LIN {X 0,Y 354.9,Z 351.278,A -85,B 0,C 180,E1 -13564.173,E2 -13564.173} C_VEL
LIN {X 0,Y 354.84,Z 351.284,A -85,B 0,C 180,E1 -13567.894,E2 -13567.894} C_VEL
LIN {X 0,Y 354.924,Z 351.273,A -85,B 0,C 180,E1 -13571.891,E2 -13571.891} C_VEL
LIN {X 0,Y 354.943,Z 351.273,A -85,B 0,C 180,E1 -13575.981,E2 -13575.981} C_VEL
LIN {X 0,Y 354.979,Z 351.267,A -85,B 0,C 180,E1 -13579.736,E2 -13579.736} C_VEL
LIN {X 0,Y 355.125,Z 351.247,A -85,B 0,C 180,E1 -13583.181,E2 -13583.181} C_VEL
LIN {X 0,Y 355.247,Z 351.234,A -85,B 0,C 180,E1 -13587.732,E2 -13587.732} C_VEL
LIN {X 0,Y 355.397,Z 351.218,A -85,B 0,C 180,E1 -13590,E2 -13590} C_VEL
LIN {X 0,Y 355.247,Z 351.234,A -85,B 0,C 180,E1 -13592.268,E2 -13592.268} C_VEL
LIN {X 0,Y 355.125,Z 351.247,A -85,B 0,C 180,E1 -13596.82,E2 -13596.82} C_VEL
LIN {X 0,Y 354.979,Z 351.267,A -85,B 0,C 180,E1 -13600.264,E2 -13600.264} C_VEL
LIN {X 0,Y 354.943,Z 351.272,A -85,B 0,C 180,E1 -13604.019,E2 -13604.019} C_VEL
LIN {X 0,Y 354.924,Z 351.274,A -85,B 0,C 180,E1 -13608.109,E2 -13608.109} C_VEL
LIN {X 0,Y 354.837,Z 351.284,A -85,B 0,C 180,E1 -13612.106,E2 -13612.106} C_VEL
LIN {X 0,Y 354.9,Z 351.278,A -85,B 0,C 180,E1 -13615.828,E2 -13615.828} C_VEL
LIN {X 0,Y 354.819,Z 351.289,A -85,B 0,C 180,E1 -13619.682,E2 -13619.682} C_VEL
LIN {X 0,Y 354.807,Z 351.289,A -85,B 0,C 180,E1 -13623.702,E2 -13623.702} C_VEL
LIN {X 0,Y 354.799,Z 351.287,A -85,B 0,C 180,E1 -13626.46,E2 -13626.46} C_VEL
LIN {X 0,Y 354.825,Z 351.288,A -85,B 0,C 180,E1 -13629.424,E2 -13629.424} C_VEL
LIN {X 0,Y 354.837,Z 351.285,A -85,B 0,C 180,E1 -13632.876,E2 -13632.876} C_VEL
LIN {X 0,Y 354.785,Z 351.289,A -85,B 0,C 180,E1 -13636.107,E2 -13636.107} C_VEL
LIN {X 0,Y 354.79,Z 351.293,A -85,B 0,C 180,E1 -13639.18,E2 -13639.18} C_VEL
LIN {X 0,Y 354.8,Z 351.285,A -85,B 0,C 180,E1 -13641.986,E2 -13641.986} C_VEL
LIN {X 0,Y 354.179,Z 351.369,A -85,B 0,C 180,E1 -13642.933,E2 -13642.933} C_VEL
LIN {X 0,Y 351.343,Z 351.731,A -85,B 0,C 180,E1 -13644.472,E2 -13644.472} C_VEL
LIN {X 0,Y 348.898,Z 352.035,A -85,B 0,C 180,E1 -13645.718,E2 -13645.718} C_VEL
LIN {X 0,Y 347.828,Z 352.162,A -85,B 0,C 180,E1 -13646.683,E2 -13646.683} C_VEL
LIN {X 0,Y 347.732,Z 352.171,A -85,B 0,C 180,E1 -13647.01,E2 -13647.01} C_VEL
LIN {X 0,Y 347.808,Z 352.163,A -85,B 0,C 180,E1 -13650.991,E2 -13650.991} C_VEL
LIN {X 0,Y 347.835,Z 352.155,A -85,B 0,C 180,E1 -13653.608,E2 -13653.608} C_VEL
LIN {X 0,Y 347.792,Z 352.16,A -85,B 0,C 180,E1 -13656.162,E2 -13656.162} C_VEL
LIN {X 0,Y 347.816,Z 352.156,A -85,B 0,C 180,E1 -13659.91,E2 -13659.91} C_VEL
LIN {X 0,Y 347.87,Z 352.152,A -85,B 0,C 180,E1 -13662.36,E2 -13662.36} C_VEL
LIN {X 0,Y 347.901,Z 352.147,A -85,B 0,C 180,E1 -13665.971,E2 -13665.971} C_VEL
LIN {X 0,Y 347.933,Z 352.143,A -85,B 0,C 180,E1 -13669.526,E2 -13669.526} C_VEL
LIN {X 0,Y 348.079,Z 352.125,A -85,B 0,C 180,E1 -13671.875,E2 -13671.875} C_VEL
LIN {X 0,Y 348.072,Z 352.127,A -85,B 0,C 180,E1 -13674.206,E2 -13674.206} C_VEL
LIN {X 0,Y 348.21,Z 352.107,A -85,B 0,C 180,E1 -13677.687,E2 -13677.687} C_VEL
LIN {X 0,Y 348.35,Z 352.092,A -85,B 0,C 180,E1 -13680,E2 -13680} C_VEL
LIN {X 0,Y 348.213,Z 352.112,A -85,B 0,C 180,E1 -13682.314,E2 -13682.314} C_VEL
LIN {X 0,Y 348.082,Z 352.125,A -85,B 0,C 180,E1 -13686.958,E2 -13686.958} C_VEL
LIN {X 0,Y 347.932,Z 352.147,A -85,B 0,C 180,E1 -13690.474,E2 -13690.474} C_VEL
LIN {X 0,Y 347.903,Z 352.15,A -85,B 0,C 180,E1 -13694.15,E2 -13694.15} C_VEL
LIN {X 0,Y 347.896,Z 352.151,A -85,B 0,C 180,E1 -13698.291,E2 -13698.291} C_VEL
LIN {X 0,Y 347.793,Z 352.161,A -85,B 0,C 180,E1 -13701.635,E2 -13701.635} C_VEL
LIN {X 0,Y 347.817,Z 352.157,A -85,B 0,C 180,E1 -13705.108,E2 -13705.108} C_VEL
LIN {X 0,Y 347.815,Z 352.16,A -85,B 0,C 180,E1 -13707.694,E2 -13707.694} C_VEL
LIN {X 0,Y 347.768,Z 352.165,A -85,B 0,C 180,E1 -13710.346,E2 -13710.346} C_VEL
LIN {X 0,Y 347.748,Z 352.166,A -85,B 0,C 180,E1 -13714.464,E2 -13714.464} C_VEL
LIN {X 0,Y 347.778,Z 352.166,A -85,B 0,C 180,E1 -13717.989,E2 -13717.989} C_VEL
LIN {X 0,Y 347.754,Z 352.169,A -85,B 0,C 180,E1 -13721.83,E2 -13721.83} C_VEL
LIN {X 0,Y 347.796,Z 352.242,A -85,B 0,C 180,E1 -13724.098,E2 -13724.098} C_VEL
LIN {X 0,Y 349.366,Z 360.314,A -85,B 0,C 180,E1 -13727.345,E2 -13727.345} C_VEL
LIN {X 0,Y 351.389,Z 370.514,A -85,B 0,C 180,E1 -13731.263,E2 -13731.263} C_VEL
LIN {X 0,Y 351.886,Z 373.789,A -85,B 0,C 180,E1 -13732.472,E2 -13732.472} C_VEL
LIN {X 0,Y 350.707,Z 383.556,A -85,B 0,C 180,E1 -13735.867,E2 -13735.867} C_VEL
LIN {X 0,Y 349.465,Z 395.227,A -85,B 0,C 180,E1 -13739.856,E2 -13739.856} C_VEL
LIN {X 0,Y 348.417,Z 406.538,A -85,B 0,C 180,E1 -13743.655,E2 -13743.655} C_VEL
LIN {X 0,Y 347.759,Z 415.945,A -85,B 0,C 180,E1 -13746.791,E2 -13746.791} C_VEL
LIN {X 0,Y 347.166,Z 427.344,A -85,B 0,C 180,E1 -13750.563,E2 -13750.563} C_VEL
LIN {X 0,Y 348.118,Z 441.877,A -85,B 0,C 180,E1 -13751.226,E2 -13751.226} C_VEL
LIN {X 0,Y 349.033,Z 455.463,A -85,B 0,C 180,E1 -13752.084,E2 -13752.084} C_VEL
LIN {X 0,Y 349.717,Z 469.057,A -85,B 0,C 180,E1 -13753.209,E2 -13753.209} C_VEL
LIN {X 0,Y 349.808,Z 475.163,A -85,B 0,C 180,E1 -13753.813,E2 -13753.813} C_VEL
LIN {X 0,Y 348.741,Z 487.264,A -85,B 0,C 180,E1 -13755.234,E2 -13755.234} C_VEL
LIN {X 0,Y 348.022,Z 496.484,A -85,B 0,C 180,E1 -13756.571,E2 -13756.571} C_VEL
LIN {X 0,Y 347.479,Z 504.803,A -85,B 0,C 180,E1 -13758.035,E2 -13758.035} C_VEL
LIN {X 0,Y 347.098,Z 512.961,A -85,B 0,C 180,E1 -13759.795,E2 -13759.795} C_VEL
LIN {X 0,Y 347.02,Z 518.533,A -85,B 0,C 180,E1 -13761.263,E2 -13761.263} C_VEL
LIN {X 0,Y 347.078,Z 523.927,A -85,B 0,C 180,E1 -13763.022,E2 -13763.022} C_VEL
LIN {X 0,Y 347.314,Z 528.073,A -85,B 0,C 180,E1 -13764.775,E2 -13764.775} C_VEL
LIN {X 0,Y 347.398,Z 531.023,A -85,B 0,C 180,E1 -13766.52,E2 -13766.52} C_VEL
LIN {X 0,Y 347.478,Z 532.411,A -85,B 0,C 180,E1 -13767.682,E2 -13767.682} C_VEL
LIN {X 0,Y 347.68,Z 533.326,A -85,B 0,C 180,E1 -13768.842,E2 -13768.842} C_VEL
LIN {X 0,Y 347.825,Z 533.775,A -85,B 0,C 180,E1 -13770,E2 -13770} C_VEL
LIN {X 0,Y 347.632,Z 533.739,A -85,B 0,C 180,E1 -13771.158,E2 -13771.158} C_VEL
LIN {X 0,Y 347.338,Z 533.253,A -85,B 0,C 180,E1 -13772.319,E2 -13772.319} C_VEL
LIN {X 0,Y 347.249,Z 532.323,A -85,B 0,C 180,E1 -13773.481,E2 -13773.481} C_VEL
LIN {X 0,Y 347.148,Z 530.952,A -85,B 0,C 180,E1 -13774.645,E2 -13774.645} C_VEL
LIN {X 0,Y 346.816,Z 527.255,A -85,B 0,C 180,E1 -13776.803,E2 -13776.803} C_VEL
LIN {X 0,Y 346.748,Z 522.608,A -85,B 0,C 180,E1 -13778.744,E2 -13778.744} C_VEL
LIN {X 0,Y 346.991,Z 516.19,A -85,B 0,C 180,E1 -13780.798,E2 -13780.798} C_VEL
LIN {X 0,Y 347.662,Z 508.139,A -85,B 0,C 180,E1 -13782.848,E2 -13782.848} C_VEL
LIN {X 0,Y 348.606,Z 499.648,A -85,B 0,C 180,E1 -13784.602,E2 -13784.602} C_VEL
LIN {X 0,Y 350.109,Z 489.465,A -85,B 0,C 180,E1 -13786.322,E2 -13786.322} C_VEL
LIN {X 0,Y 351.852,Z 478.234,A -85,B 0,C 180,E1 -13787.885,E2 -13787.885} C_VEL
LIN {X 0,Y 352.667,Z 465.91,A -85,B 0,C 180,E1 -13789.348,E2 -13789.348} C_VEL
LIN {X 0,Y 353.333,Z 454.376,A -85,B 0,C 180,E1 -13790.502,E2 -13790.502} C_VEL
LIN {X 0,Y 352.981,Z 441.435,A -85,B 0,C 180,E1 -13791.675,E2 -13791.675} C_VEL
LIN {X 0,Y 351.394,Z 428.535,A -85,B 0,C 180,E1 -13792.778,E2 -13792.778} C_VEL
LIN {X 0,Y 348.621,Z 415.219,A -85,B 0,C 180,E1 -13793.896,E2 -13793.896} C_VEL
LIN {X 0,Y 347.813,Z 411.035,A -85,B 0,C 180,E1 -13794.239,E2 -13794.239} C_VEL
LIN {X 0,Y 348.505,Z 400.916,A -85,B 0,C 180,E1 -13797.634,E2 -13797.634} C_VEL
LIN {X 0,Y 349.397,Z 391.787,A -85,B 0,C 180,E1 -13800.859,E2 -13800.859} C_VEL
LIN {X 0,Y 350.778,Z 381.485,A -85,B 0,C 180,E1 -13804.769,E2 -13804.769} C_VEL
LIN {X 0,Y 352.109,Z 374.816,A -85,B 0,C 180,E1 -13807.503,E2 -13807.503} C_VEL
LIN {X 0,Y 351.539,Z 370.215,A -85,B 0,C 180,E1 -13809.773,E2 -13809.773} C_VEL
LIN {X 0,Y 350.498,Z 364.605,A -85,B 0,C 180,E1 -13812.981,E2 -13812.981} C_VEL
LIN {X 0,Y 349.381,Z 359.714,A -85,B 0,C 180,E1 -13816.399,E2 -13816.399} C_VEL
LIN {X 0,Y 348.924,Z 357.382,A -85,B 0,C 180,E1 -13818.342,E2 -13818.342} C_VEL
LIN {X 0,Y 348.163,Z 353.938,A -85,B 0,C 180,E1 -13821.93,E2 -13821.93} C_VEL
LIN {X 0,Y 347.798,Z 352.163,A -85,B 0,C 180,E1 -13824.482,E2 -13824.482} C_VEL
LIN {X 0,Y 347.748,Z 352.166,A -85,B 0,C 180,E1 -13828.3,E2 -13828.3} C_VEL
LIN {X 0,Y 347.808,Z 352.161,A -85,B 0,C 180,E1 -13830.99,E2 -13830.99} C_VEL
LIN {X 0,Y 347.835,Z 352.156,A -85,B 0,C 180,E1 -13833.608,E2 -13833.608} C_VEL
LIN {X 0,Y 347.843,Z 352.27,A -85,B 0,C 180,E1 -13835.277,E2 -13835.277} C_VEL
LIN {X 0,Y 348.889,Z 355.097,A -85,B 0,C 180,E1 -13835.649,E2 -13835.649} C_VEL
LIN {X 0,Y 349.761,Z 356.218,A -85,B 0,C 180,E1 -13835.875,E2 -13835.875} C_VEL
LIN {X 0,Y 355.432,Z 368.089,A -85,B 0,C 180,E1 -13837.74,E2 -13837.74} C_VEL
LIN {X 0,Y 358.834,Z 377.479,A -85,B 0,C 180,E1 -13839.196,E2 -13839.196} C_VEL
LIN {X 0,Y 359.888,Z 381.885,A -85,B 0,C 180,E1 -13839.87,E2 -13839.87} C_VEL
LIN {X 0,Y 358.454,Z 392.191,A -85,B 0,C 180,E1 -13841.125,E2 -13841.125} C_VEL
LIN {X 0,Y 356.868,Z 401.532,A -85,B 0,C 180,E1 -13842.523,E2 -13842.523} C_VEL
LIN {X 0,Y 355.192,Z 410.63,A -85,B 0,C 180,E1 -13844.213,E2 -13844.213} C_VEL
LIN {X 0,Y 353.658,Z 418.033,A -85,B 0,C 180,E1 -13845.91,E2 -13845.91} C_VEL
LIN {X 0,Y 352.237,Z 424.697,A -85,B 0,C 180,E1 -13847.871,E2 -13847.871} C_VEL
LIN {X 0,Y 351.047,Z 429.307,A -85,B 0,C 180,E1 -13849.62,E2 -13849.62} C_VEL
LIN {X 0,Y 350.364,Z 431.687,A -85,B 0,C 180,E1 -13850.765,E2 -13850.765} C_VEL
LIN {X 0,Y 349.862,Z 433.615,A -85,B 0,C 180,E1 -13851.916,E2 -13851.916} C_VEL
LIN {X 0,Y 349.316,Z 435.152,A -85,B 0,C 180,E1 -13853.066,E2 -13853.066} C_VEL
LIN {X 0,Y 348.965,Z 436.221,A -85,B 0,C 180,E1 -13854.22,E2 -13854.22} C_VEL
LIN {X 0,Y 348.368,Z 437.149,A -85,B 0,C 180,E1 -13856.53,E2 -13856.53} C_VEL
LIN {X 0,Y 348.165,Z 437.026,A -85,B 0,C 180,E1 -13857.686,E2 -13857.686} C_VEL
LIN {X 0,Y 348.011,Z 436.465,A -85,B 0,C 180,E1 -13858.843,E2 -13858.843} C_VEL
LIN {X 0,Y 347.933,Z 435.505,A -85,B 0,C 180,E1 -13860,E2 -13860} C_VEL
LIN {X 0,Y 347.774,Z 434.173,A -85,B 0,C 180,E1 -13861.158,E2 -13861.158} C_VEL
LIN {X 0,Y 347.754,Z 431.335,A -85,B 0,C 180,E1 -13862.896,E2 -13862.896} C_VEL
LIN {X 0,Y 347.898,Z 427.484,A -85,B 0,C 180,E1 -13864.635,E2 -13864.635} C_VEL
LIN {X 0,Y 348.373,Z 422.514,A -85,B 0,C 180,E1 -13866.37,E2 -13866.37} C_VEL
LIN {X 0,Y 348.729,Z 416.322,A -85,B 0,C 180,E1 -13868.11,E2 -13868.11} C_VEL
LIN {X 0,Y 349.305,Z 408.669,A -85,B 0,C 180,E1 -13869.846,E2 -13869.846} C_VEL
LIN {X 0,Y 349.935,Z 399.29,A -85,B 0,C 180,E1 -13871.586,E2 -13871.586} C_VEL
LIN {X 0,Y 350.781,Z 388.629,A -85,B 0,C 180,E1 -13873.173,E2 -13873.173} C_VEL
LIN {X 0,Y 351.477,Z 377.977,A -85,B 0,C 180,E1 -13874.474,E2 -13874.474} C_VEL
LIN {X 0,Y 351.792,Z 367.9,A -85,B 0,C 180,E1 -13875.497,E2 -13875.497} C_VEL
LIN {X 0,Y 348.726,Z 355.743,A -85,B 0,C 180,E1 -13876.614,E2 -13876.614} C_VEL
LIN {X 0,Y 347.872,Z 352.153,A -85,B 0,C 180,E1 -13876.921,E2 -13876.921} C_VEL
LIN {X 0,Y 347.814,Z 352.157,A -85,B 0,C 180,E1 -13880.09,E2 -13880.09} C_VEL
LIN {X 0,Y 347.791,Z 352.16,A -85,B 0,C 180,E1 -13883.838,E2 -13883.838} C_VEL
LIN {X 0,Y 347.854,Z 352.156,A -85,B 0,C 180,E1 -13887.255,E2 -13887.255} C_VEL
LIN {X 0,Y 347.766,Z 352.164,A -85,B 0,C 180,E1 -13890.346,E2 -13890.346} C_VEL
LIN {X 0,Y 347.746,Z 352.167,A -85,B 0,C 180,E1 -13894.464,E2 -13894.464} C_VEL
LIN {X 0,Y 347.778,Z 352.161,A -85,B 0,C 180,E1 -13897.989,E2 -13897.989} C_VEL
LIN {X 0,Y 347.768,Z 352.163,A -85,B 0,C 180,E1 -13901.828,E2 -13901.828} C_VEL
LIN {X 0,Y 347.768,Z 352.166,A -85,B 0,C 180,E1 -13905.016,E2 -13905.016} C_VEL
LIN {X 0,Y 347.752,Z 352.168,A -85,B 0,C 180,E1 -13908.397,E2 -13908.397} C_VEL
LIN {X 0,Y 347.777,Z 352.162,A -85,B 0,C 180,E1 -13912.01,E2 -13912.01} C_VEL
LIN {X 0,Y 347.745,Z 352.165,A -85,B 0,C 180,E1 -13915.536,E2 -13915.536} C_VEL
LIN {X 0,Y 347.746,Z 352.169,A -85,B 0,C 180,E1 -13918.3,E2 -13918.3} C_VEL
LIN {X 0,Y 347.779,Z 352.163,A -85,B 0,C 180,E1 -13920.988,E2 -13920.988} C_VEL
LIN {X 0,Y 347.831,Z 352.155,A -85,B 0,C 180,E1 -13923.608,E2 -13923.608} C_VEL
LIN {X 0,Y 347.79,Z 352.164,A -85,B 0,C 180,E1 -13926.162,E2 -13926.162} C_VEL
LIN {X 0,Y 347.828,Z 352.157,A -85,B 0,C 180,E1 -13929.91,E2 -13929.91} C_VEL
LIN {X 0,Y 347.868,Z 352.155,A -85,B 0,C 180,E1 -13932.359,E2 -13932.359} C_VEL
LIN {X 0,Y 347.898,Z 352.15,A -85,B 0,C 180,E1 -13935.971,E2 -13935.971} C_VEL
LIN {X 0,Y 347.929,Z 352.144,A -85,B 0,C 180,E1 -13939.526,E2 -13939.526} C_VEL
LIN {X 0,Y 348.091,Z 352.123,A -85,B 0,C 180,E1 -13943.042,E2 -13943.042} C_VEL
LIN {X 0,Y 348.209,Z 352.11,A -85,B 0,C 180,E1 -13947.687,E2 -13947.687} C_VEL
LIN {X 0,Y 348.346,Z 352.096,A -85,B 0,C 180,E1 -13950,E2 -13950} C_VEL
LIN {X 0,Y 348.21,Z 352.11,A -85,B 0,C 180,E1 -13952.314,E2 -13952.314} C_VEL
LIN {X 0,Y 348.091,Z 352.123,A -85,B 0,C 180,E1 -13956.958,E2 -13956.958} C_VEL
LIN {X 0,Y 347.93,Z 352.144,A -85,B 0,C 180,E1 -13960.475,E2 -13960.475} C_VEL
LIN {X 0,Y 347.899,Z 352.149,A -85,B 0,C 180,E1 -13964.15,E2 -13964.15} C_VEL
LIN {X 0,Y 347.892,Z 352.148,A -85,B 0,C 180,E1 -13968.291,E2 -13968.291} C_VEL
LIN {X 0,Y 347.791,Z 352.165,A -85,B 0,C 180,E1 -13971.636,E2 -13971.636} C_VEL
LIN {X 0,Y 347.813,Z 352.159,A -85,B 0,C 180,E1 -13975.109,E2 -13975.109} C_VEL
LIN {X 0,Y 347.809,Z 352.162,A -85,B 0,C 180,E1 -13977.694,E2 -13977.694} C_VEL
LIN {X 0,Y 347.75,Z 352.165,A -85,B 0,C 180,E1 -13980.348,E2 -13980.348} C_VEL
LIN {X 0,Y 347.749,Z 352.166,A -85,B 0,C 180,E1 -13984.044,E2 -13984.044} C_VEL
LIN {X 0,Y 347.763,Z 352.169,A -85,B 0,C 180,E1 -13987.321,E2 -13987.321} C_VEL
LIN {X 0,Y 347.795,Z 352.16,A -85,B 0,C 180,E1 -13990.289,E2 -13990.289} C_VEL
LIN {X 0,Y 347.788,Z 352.165,A -85,B 0,C 180,E1 -13993.399,E2 -13993.399} C_VEL
LIN {X 0,Y 347.731,Z 352.169,A -85,B 0,C 180,E1 -13996.686,E2 -13996.686} C_VEL
LIN {X 0,Y 347.749,Z 352.165,A -85,B 0,C 180,E1 -14000.173,E2 -14000.173} C_VEL
LIN {X 0,Y 347.764,Z 352.165,A -85,B 0,C 180,E1 -14002.68,E2 -14002.68} C_VEL
LIN {X 0,Y 347.751,Z 352.165,A -85,B 0,C 180,E1 -14005.957,E2 -14005.957} C_VEL
LIN {X 0,Y 347.732,Z 352.171,A -85,B 0,C 180,E1 -14007.01,E2 -14007.01} C_VEL
LIN {X 0,Y 347.039,Z 352.254,A -85,B 0,C 180,E1 -14007.978,E2 -14007.978} C_VEL
LIN {X 0,Y 344.186,Z 352.61,A -85,B 0,C 180,E1 -14009.553,E2 -14009.553} C_VEL
LIN {X 0,Y 341.809,Z 352.91,A -85,B 0,C 180,E1 -14010.828,E2 -14010.828} C_VEL
LIN {X 0,Y 340.822,Z 353.028,A -85,B 0,C 180,E1 -14011.815,E2 -14011.815} C_VEL
LIN {X 0,Y 340.758,Z 353.036,A -85,B 0,C 180,E1 -14012.148,E2 -14012.148} C_VEL
LIN {X 0,Y 340.759,Z 353.036,A -85,B 0,C 180,E1 -14015.639,E2 -14015.639} C_VEL
LIN {X 0,Y 340.756,Z 353.037,A -85,B 0,C 180,E1 -14019.475,E2 -14019.475} C_VEL
LIN {X 0,Y 340.861,Z 353.023,A -85,B 0,C 180,E1 -14021.985,E2 -14021.985} C_VEL
LIN {X 0,Y 340.873,Z 353.022,A -85,B 0,C 180,E1 -14025.705,E2 -14025.705} C_VEL
LIN {X 0,Y 340.876,Z 353.022,A -85,B 0,C 180,E1 -14029.307,E2 -14029.307} C_VEL
LIN {X 0,Y 341.081,Z 352.999,A -85,B 0,C 180,E1 -14032.899,E2 -14032.899} C_VEL
LIN {X 0,Y 341.172,Z 352.984,A -85,B 0,C 180,E1 -14037.639,E2 -14037.639} C_VEL
LIN {X 0,Y 341.3,Z 352.97,A -85,B 0,C 180,E1 -14040,E2 -14040} C_VEL
LIN {X 0,Y 341.175,Z 352.989,A -85,B 0,C 180,E1 -14042.361,E2 -14042.361} C_VEL
LIN {X 0,Y 341.05,Z 353,A -85,B 0,C 180,E1 -14047.103,E2 -14047.103} C_VEL
LIN {X 0,Y 340.875,Z 353.024,A -85,B 0,C 180,E1 -14050.694,E2 -14050.694} C_VEL
LIN {X 0,Y 340.867,Z 353.027,A -85,B 0,C 180,E1 -14054.325,E2 -14054.325} C_VEL
LIN {X 0,Y 340.842,Z 353.029,A -85,B 0,C 180,E1 -14058.467,E2 -14058.467} C_VEL
LIN {X 0,Y 340.758,Z 353.039,A -85,B 0,C 180,E1 -14061.857,E2 -14061.857} C_VEL
LIN {X 0,Y 340.777,Z 353.036,A -85,B 0,C 180,E1 -14065.664,E2 -14065.664} C_VEL
LIN {X 0,Y 340.745,Z 353.041,A -85,B 0,C 180,E1 -14068.32,E2 -14068.32} C_VEL
LIN {X 0,Y 340.708,Z 353.042,A -85,B 0,C 180,E1 -14071.044,E2 -14071.044} C_VEL
LIN {X 0,Y 340.722,Z 353.041,A -85,B 0,C 180,E1 -14075.279,E2 -14075.279} C_VEL
LIN {X 0,Y 340.714,Z 353.043,A -85,B 0,C 180,E1 -14078.386,E2 -14078.386} C_VEL
LIN {X 0,Y 340.705,Z 353.047,A -85,B 0,C 180,E1 -14082.046,E2 -14082.046} C_VEL
LIN {X 0,Y 340.741,Z 353.14,A -85,B 0,C 180,E1 -14083.835,E2 -14083.835} C_VEL
LIN {X 0,Y 342.524,Z 362.377,A -85,B 0,C 180,E1 -14087.618,E2 -14087.618} C_VEL
LIN {X 0,Y 344.203,Z 370.698,A -85,B 0,C 180,E1 -14090.886,E2 -14090.886} C_VEL
LIN {X 0,Y 344.84,Z 374.465,A -85,B 0,C 180,E1 -14092.308,E2 -14092.308} C_VEL
LIN {X 0,Y 343.679,Z 384.226,A -85,B 0,C 180,E1 -14095.781,E2 -14095.781} C_VEL
LIN {X 0,Y 342.485,Z 394.939,A -85,B 0,C 180,E1 -14099.527,E2 -14099.527} C_VEL
LIN {X 0,Y 341.497,Z 405.244,A -85,B 0,C 180,E1 -14103.079,E2 -14103.079} C_VEL
LIN {X 0,Y 340.635,Z 416.46,A -85,B 0,C 180,E1 -14106.92,E2 -14106.92} C_VEL
LIN {X 0,Y 340.112,Z 426.416,A -85,B 0,C 180,E1 -14110.301,E2 -14110.301} C_VEL
LIN {X 0,Y 341.079,Z 442.102,A -85,B 0,C 180,E1 -14111.056,E2 -14111.056} C_VEL
LIN {X 0,Y 341.969,Z 455.589,A -85,B 0,C 180,E1 -14111.956,E2 -14111.956} C_VEL
LIN {X 0,Y 342.601,Z 467.846,A -85,B 0,C 180,E1 -14113.003,E2 -14113.003} C_VEL
LIN {X 0,Y 342.713,Z 475.376,A -85,B 0,C 180,E1 -14113.775,E2 -14113.775} C_VEL
LIN {X 0,Y 341.665,Z 487.006,A -85,B 0,C 180,E1 -14115.192,E2 -14115.192} C_VEL
LIN {X 0,Y 340.926,Z 496.262,A -85,B 0,C 180,E1 -14116.59,E2 -14116.59} C_VEL
LIN {X 0,Y 340.391,Z 504.438,A -85,B 0,C 180,E1 -14118.084,E2 -14118.084} C_VEL
LIN {X 0,Y 340.024,Z 512.478,A -85,B 0,C 180,E1 -14119.881,E2 -14119.881} C_VEL
LIN {X 0,Y 339.999,Z 518.948,A -85,B 0,C 180,E1 -14121.68,E2 -14121.68} C_VEL
LIN {X 0,Y 340.105,Z 524.358,A -85,B 0,C 180,E1 -14123.623,E2 -14123.623} C_VEL
LIN {X 0,Y 340.332,Z 527.843,A -85,B 0,C 180,E1 -14125.262,E2 -14125.262} C_VEL
LIN {X 0,Y 340.382,Z 529.72,A -85,B 0,C 180,E1 -14126.449,E2 -14126.449} C_VEL
LIN {X 0,Y 340.483,Z 531.149,A -85,B 0,C 180,E1 -14127.634,E2 -14127.634} C_VEL
LIN {X 0,Y 340.676,Z 532.141,A -85,B 0,C 180,E1 -14128.818,E2 -14128.818} C_VEL
LIN {X 0,Y 340.813,Z 532.631,A -85,B 0,C 180,E1 -14130,E2 -14130} C_VEL
LIN {X 0,Y 340.601,Z 532.626,A -85,B 0,C 180,E1 -14131.182,E2 -14131.182} C_VEL
LIN {X 0,Y 340.303,Z 532.179,A -85,B 0,C 180,E1 -14132.367,E2 -14132.367} C_VEL
LIN {X 0,Y 340.198,Z 531.321,A -85,B 0,C 180,E1 -14133.553,E2 -14133.553} C_VEL
LIN {X 0,Y 340.079,Z 529.987,A -85,B 0,C 180,E1 -14134.742,E2 -14134.742} C_VEL
LIN {X 0,Y 339.739,Z 526.641,A -85,B 0,C 180,E1 -14136.805,E2 -14136.805} C_VEL
LIN {X 0,Y 339.679,Z 521.815,A -85,B 0,C 180,E1 -14138.927,E2 -14138.927} C_VEL
LIN {X 0,Y 339.965,Z 515.568,A -85,B 0,C 180,E1 -14141.024,E2 -14141.024} C_VEL
LIN {X 0,Y 340.683,Z 507.658,A -85,B 0,C 180,E1 -14143.116,E2 -14143.116} C_VEL
LIN {X 0,Y 341.733,Z 499.139,A -85,B 0,C 180,E1 -14144.95,E2 -14144.95} C_VEL
LIN {X 0,Y 343.284,Z 489.47,A -85,B 0,C 180,E1 -14146.656,E2 -14146.656} C_VEL
LIN {X 0,Y 345.183,Z 477.464,A -85,B 0,C 180,E1 -14148.396,E2 -14148.396} C_VEL
LIN {X 0,Y 346.158,Z 465.409,A -85,B 0,C 180,E1 -14149.881,E2 -14149.881} C_VEL
LIN {X 0,Y 346.901,Z 453.696,A -85,B 0,C 180,E1 -14151.106,E2 -14151.106} C_VEL
LIN {X 0,Y 346.586,Z 442.117,A -85,B 0,C 180,E1 -14152.224,E2 -14152.224} C_VEL
LIN {X 0,Y 345.233,Z 429.937,A -85,B 0,C 180,E1 -14153.348,E2 -14153.348} C_VEL
LIN {X 0,Y 342.129,Z 414.017,A -85,B 0,C 180,E1 -14154.786,E2 -14154.786} C_VEL
LIN {X 0,Y 341.004,Z 409.581,A -85,B 0,C 180,E1 -14155.198,E2 -14155.198} C_VEL
LIN {X 0,Y 340.97,Z 408.959,A -85,B 0,C 180,E1 -14155.28,E2 -14155.28} C_VEL
LIN {X 0,Y 341.79,Z 398.636,A -85,B 0,C 180,E1 -14158.896,E2 -14158.896} C_VEL
LIN {X 0,Y 342.826,Z 389.705,A -85,B 0,C 180,E1 -14162.209,E2 -14162.209} C_VEL
LIN {X 0,Y 344.513,Z 379.586,A -85,B 0,C 180,E1 -14166.271,E2 -14166.271} C_VEL
LIN {X 0,Y 345.246,Z 376.385,A -85,B 0,C 180,E1 -14167.64,E2 -14167.64} C_VEL
LIN {X 0,Y 344.659,Z 371.814,A -85,B 0,C 180,E1 -14169.965,E2 -14169.965} C_VEL
LIN {X 0,Y 343.814,Z 367.247,A -85,B 0,C 180,E1 -14172.618,E2 -14172.618} C_VEL
LIN {X 0,Y 342.763,Z 362.561,A -85,B 0,C 180,E1 -14175.86,E2 -14175.86} C_VEL
LIN {X 0,Y 341.875,Z 358.319,A -85,B 0,C 180,E1 -14179.519,E2 -14179.519} C_VEL
LIN {X 0,Y 341.437,Z 356.176,A -85,B 0,C 180,E1 -14181.865,E2 -14181.865} C_VEL
LIN {X 0,Y 340.828,Z 353.656,A -85,B 0,C 180,E1 -14185.57,E2 -14185.57} C_VEL
LIN {X 0,Y 340.712,Z 353.042,A -85,B 0,C 180,E1 -14186.864,E2 -14186.864} C_VEL
LIN {X 0,Y 340.778,Z 353.033,A -85,B 0,C 180,E1 -14190.332,E2 -14190.332} C_VEL
LIN {X 0,Y 340.77,Z 353.038,A -85,B 0,C 180,E1 -14194.13,E2 -14194.13} C_VEL
LIN {X 0,Y 341.257,Z 354.834,A -85,B 0,C 180,E1 -14194.374,E2 -14194.374} C_VEL
LIN {X 0,Y 343.025,Z 357.39,A -85,B 0,C 180,E1 -14194.882,E2 -14194.882} C_VEL
LIN {X 0,Y 348.655,Z 368.859,A -85,B 0,C 180,E1 -14196.847,E2 -14196.847} C_VEL
LIN {X 0,Y 352.112,Z 377.872,A -85,B 0,C 180,E1 -14198.348,E2 -14198.348} C_VEL
LIN {X 0,Y 353.825,Z 384.581,A -85,B 0,C 180,E1 -14199.432,E2 -14199.432} C_VEL
LIN {X 0,Y 352.139,Z 394.973,A -85,B 0,C 180,E1 -14200.773,E2 -14200.773} C_VEL
LIN {X 0,Y 350.171,Z 405.658,A -85,B 0,C 180,E1 -14202.479,E2 -14202.479} C_VEL
LIN {X 0,Y 348.377,Z 414.184,A -85,B 0,C 180,E1 -14204.196,E2 -14204.196} C_VEL
LIN {X 0,Y 346.79,Z 421.072,A -85,B 0,C 180,E1 -14205.925,E2 -14205.925} C_VEL
LIN {X 0,Y 345.536,Z 426.547,A -85,B 0,C 180,E1 -14207.652,E2 -14207.652} C_VEL
LIN {X 0,Y 344.261,Z 430.973,A -85,B 0,C 180,E1 -14209.413,E2 -14209.413} C_VEL
LIN {X 0,Y 343.559,Z 433.259,A -85,B 0,C 180,E1 -14210.581,E2 -14210.581} C_VEL
LIN {X 0,Y 343.017,Z 435.102,A -85,B 0,C 180,E1 -14211.754,E2 -14211.754} C_VEL
LIN {X 0,Y 342.433,Z 436.548,A -85,B 0,C 180,E1 -14212.926,E2 -14212.926} C_VEL
LIN {X 0,Y 341.674,Z 438.125,A -85,B 0,C 180,E1 -14215.28,E2 -14215.28} C_VEL
LIN {X 0,Y 341.38,Z 438.342,A -85,B 0,C 180,E1 -14216.459,E2 -14216.459} C_VEL
LIN {X 0,Y 341.156,Z 438.132,A -85,B 0,C 180,E1 -14217.638,E2 -14217.638} C_VEL
LIN {X 0,Y 340.91,Z 436.486,A -85,B 0,C 180,E1 -14220,E2 -14220} C_VEL
LIN {X 0,Y 340.748,Z 435.083,A -85,B 0,C 180,E1 -14221.182,E2 -14221.182} C_VEL
LIN {X 0,Y 340.72,Z 432.144,A -85,B 0,C 180,E1 -14222.956,E2 -14222.956} C_VEL
LIN {X 0,Y 340.873,Z 428.189,A -85,B 0,C 180,E1 -14224.73,E2 -14224.73} C_VEL
LIN {X 0,Y 341.361,Z 423.089,A -85,B 0,C 180,E1 -14226.502,E2 -14226.502} C_VEL
LIN {X 0,Y 341.877,Z 415.678,A -85,B 0,C 180,E1 -14228.538,E2 -14228.538} C_VEL
LIN {X 0,Y 342.412,Z 407.652,A -85,B 0,C 180,E1 -14230.316,E2 -14230.316} C_VEL
LIN {X 0,Y 343.121,Z 397.528,A -85,B 0,C 180,E1 -14232.119,E2 -14232.119} C_VEL
LIN {X 0,Y 343.896,Z 387.391,A -85,B 0,C 180,E1 -14233.593,E2 -14233.593} C_VEL
LIN {X 0,Y 344.631,Z 376.16,A -85,B 0,C 180,E1 -14234.919,E2 -14234.919} C_VEL
LIN {X 0,Y 344.728,Z 368.818,A -85,B 0,C 180,E1 -14235.668,E2 -14235.668} C_VEL
LIN {X 0,Y 341.683,Z 356.599,A -85,B 0,C 180,E1 -14236.813,E2 -14236.813} C_VEL
LIN {X 0,Y 340.838,Z 353.031,A -85,B 0,C 180,E1 -14237.126,E2 -14237.126} C_VEL
LIN {X 0,Y 340.755,Z 353.037,A -85,B 0,C 180,E1 -14240.525,E2 -14240.525} C_VEL
LIN {X 0,Y 340.759,Z 353.036,A -85,B 0,C 180,E1 -14244.361,E2 -14244.361} C_VEL
LIN {X 0,Y 340.781,Z 353.035,A -85,B 0,C 180,E1 -14247.526,E2 -14247.526} C_VEL
LIN {X 0,Y 340.706,Z 353.048,A -85,B 0,C 180,E1 -14251.044,E2 -14251.044} C_VEL
LIN {X 0,Y 340.72,Z 353.043,A -85,B 0,C 180,E1 -14255.278,E2 -14255.278} C_VEL
LIN {X 0,Y 340.72,Z 353.042,A -85,B 0,C 180,E1 -14258.388,E2 -14258.388} C_VEL
LIN {X 0,Y 340.734,Z 353.039,A -85,B 0,C 180,E1 -14262.052,E2 -14262.052} C_VEL
LIN {X 0,Y 340.685,Z 353.046,A -85,B 0,C 180,E1 -14265.461,E2 -14265.461} C_VEL
LIN {X 0,Y 340.687,Z 353.05,A -85,B 0,C 180,E1 -14268.69,E2 -14268.69} C_VEL
LIN {X 0,Y 340.736,Z 353.039,A -85,B 0,C 180,E1 -14271.773,E2 -14271.773} C_VEL
LIN {X 0,Y 340.723,Z 353.04,A -85,B 0,C 180,E1 -14275.595,E2 -14275.595} C_VEL
LIN {X 0,Y 340.698,Z 353.045,A -85,B 0,C 180,E1 -14278.955,E2 -14278.955} C_VEL
LIN {X 0,Y 340.804,Z 353.031,A -85,B 0,C 180,E1 -14283.02,E2 -14283.02} C_VEL
LIN {X 0,Y 340.731,Z 353.04,A -85,B 0,C 180,E1 -14286.927,E2 -14286.927} C_VEL
LIN {X 0,Y 340.8,Z 353.032,A -85,B 0,C 180,E1 -14290.734,E2 -14290.734} C_VEL
LIN {X 0,Y 340.787,Z 353.032,A -85,B 0,C 180,E1 -14293.219,E2 -14293.219} C_VEL
LIN {X 0,Y 340.845,Z 353.026,A -85,B 0,C 180,E1 -14296.89,E2 -14296.89} C_VEL
LIN {X 0,Y 340.914,Z 353.019,A -85,B 0,C 180,E1 -14300.507,E2 -14300.507} C_VEL
LIN {X 0,Y 341.059,Z 352.999,A -85,B 0,C 180,E1 -14302.898,E2 -14302.898} C_VEL
LIN {X 0,Y 341.171,Z 352.987,A -85,B 0,C 180,E1 -14307.639,E2 -14307.639} C_VEL
LIN {X 0,Y 341.296,Z 352.974,A -85,B 0,C 180,E1 -14310,E2 -14310} C_VEL
LIN {X 0,Y 341.171,Z 352.987,A -85,B 0,C 180,E1 -14312.361,E2 -14312.361} C_VEL
LIN {X 0,Y 341.059,Z 352.999,A -85,B 0,C 180,E1 -14317.102,E2 -14317.102} C_VEL
LIN {X 0,Y 340.872,Z 353.022,A -85,B 0,C 180,E1 -14320.694,E2 -14320.694} C_VEL
LIN {X 0,Y 340.864,Z 353.024,A -85,B 0,C 180,E1 -14324.325,E2 -14324.325} C_VEL
LIN {X 0,Y 340.839,Z 353.026,A -85,B 0,C 180,E1 -14328.467,E2 -14328.467} C_VEL
LIN {X 0,Y 340.754,Z 353.04,A -85,B 0,C 180,E1 -14331.857,E2 -14331.857} C_VEL
LIN {X 0,Y 340.773,Z 353.039,A -85,B 0,C 180,E1 -14335.665,E2 -14335.665} C_VEL
LIN {X 0,Y 340.729,Z 353.04,A -85,B 0,C 180,E1 -14338.321,E2 -14338.321} C_VEL
LIN {X 0,Y 340.699,Z 353.045,A -85,B 0,C 180,E1 -14341.045,E2 -14341.045} C_VEL
LIN {X 0,Y 340.719,Z 353.045,A -85,B 0,C 180,E1 -14345.279,E2 -14345.279} C_VEL
LIN {X 0,Y 340.713,Z 353.041,A -85,B 0,C 180,E1 -14348.387,E2 -14348.387} C_VEL
LIN {X 0,Y 340.727,Z 353.045,A -85,B 0,C 180,E1 -14351.304,E2 -14351.304} C_VEL
LIN {X 0,Y 340.723,Z 353.041,A -85,B 0,C 180,E1 -14354.533,E2 -14354.533} C_VEL
LIN {X 0,Y 340.688,Z 353.046,A -85,B 0,C 180,E1 -14358.691,E2 -14358.691} C_VEL
LIN {X 0,Y 340.735,Z 353.039,A -85,B 0,C 180,E1 -14361.773,E2 -14361.773} C_VEL
LIN {X 0,Y 340.725,Z 353.041,A -85,B 0,C 180,E1 -14365.596,E2 -14365.596} C_VEL
LIN {X 0,Y 340.707,Z 353.048,A -85,B 0,C 180,E1 -14368.956,E2 -14368.956} C_VEL
LIN {X 0,Y 340.758,Z 353.036,A -85,B 0,C 180,E1 -14372.148,E2 -14372.148} C_VEL
LIN {X 0,Y 340.121,Z 353.119,A -85,B 0,C 180,E1 -14373.135,E2 -14373.135} C_VEL
LIN {X 0,Y 337.231,Z 353.479,A -85,B 0,C 180,E1 -14374.738,E2 -14374.738} C_VEL
LIN {X 0,Y 334.774,Z 353.781,A -85,B 0,C 180,E1 -14376.037,E2 -14376.037} C_VEL
LIN {X 0,Y 333.744,Z 353.914,A -85,B 0,C 180,E1 -14377.043,E2 -14377.043} C_VEL
LIN {X 0,Y 333.674,Z 353.916,A -85,B 0,C 180,E1 -14377.384,E2 -14377.384} C_VEL
LIN {X 0,Y 333.797,Z 353.903,A -85,B 0,C 180,E1 -14381.59,E2 -14381.59} C_VEL
LIN {X 0,Y 333.812,Z 353.901,A -85,B 0,C 180,E1 -14385.577,E2 -14385.577} C_VEL
LIN {X 0,Y 333.838,Z 353.9,A -85,B 0,C 180,E1 -14389.078,E2 -14389.078} C_VEL
LIN {X 0,Y 334.03,Z 353.878,A -85,B 0,C 180,E1 -14392.748,E2 -14392.748} C_VEL
LIN {X 0,Y 333.813,Z 353.902,A -85,B 0,C 180,E1 -14395.169,E2 -14395.169} C_VEL
LIN {X 0,Y 334.109,Z 353.864,A -85,B 0,C 180,E1 -14397.589,E2 -14397.589} C_VEL
LIN {X 0,Y 334.251,Z 353.848,A -85,B 0,C 180,E1 -14400,E2 -14400} C_VEL
LIN {X 0,Y 334.112,Z 353.869,A -85,B 0,C 180,E1 -14402.411,E2 -14402.411} C_VEL
LIN {X 0,Y 334.013,Z 353.879,A -85,B 0,C 180,E1 -14406.039,E2 -14406.039} C_VEL
LIN {X 0,Y 333.853,Z 353.897,A -85,B 0,C 180,E1 -14409.696,E2 -14409.696} C_VEL
LIN {X 0,Y 333.801,Z 353.902,A -85,B 0,C 180,E1 -14413.391,E2 -14413.391} C_VEL
LIN {X 0,Y 333.751,Z 353.908,A -85,B 0,C 180,E1 -14417.146,E2 -14417.146} C_VEL
LIN {X 0,Y 333.744,Z 353.911,A -85,B 0,C 180,E1 -14419.69,E2 -14419.69} C_VEL
LIN {X 0,Y 333.696,Z 353.92,A -85,B 0,C 180,E1 -14422.278,E2 -14422.278} C_VEL
LIN {X 0,Y 333.74,Z 353.914,A -85,B 0,C 180,E1 -14426.246,E2 -14426.246} C_VEL
LIN {X 0,Y 333.715,Z 353.913,A -85,B 0,C 180,E1 -14428.972,E2 -14428.972} C_VEL
LIN {X 0,Y 333.65,Z 353.922,A -85,B 0,C 180,E1 -14432.588,E2 -14432.588} C_VEL
LIN {X 0,Y 333.68,Z 353.921,A -85,B 0,C 180,E1 -14436.139,E2 -14436.139} C_VEL
LIN {X 0,Y 333.651,Z 353.922,A -85,B 0,C 180,E1 -14439.192,E2 -14439.192} C_VEL
LIN {X 0,Y 333.666,Z 353.924,A -85,B 0,C 180,E1 -14443.213,E2 -14443.213} C_VEL
LIN {X 0,Y 333.697,Z 354.141,A -85,B 0,C 180,E1 -14443.617,E2 -14443.617} C_VEL
LIN {X 0,Y 335.366,Z 362.616,A -85,B 0,C 180,E1 -14447.178,E2 -14447.178} C_VEL
LIN {X 0,Y 337.228,Z 371.946,A -85,B 0,C 180,E1 -14450.913,E2 -14450.913} C_VEL
LIN {X 0,Y 337.798,Z 375.375,A -85,B 0,C 180,E1 -14452.242,E2 -14452.242} C_VEL
LIN {X 0,Y 336.65,Z 384.836,A -85,B 0,C 180,E1 -14455.69,E2 -14455.69} C_VEL
LIN {X 0,Y 335.31,Z 396.333,A -85,B 0,C 180,E1 -14459.799,E2 -14459.799} C_VEL
LIN {X 0,Y 334.193,Z 407.642,A -85,B 0,C 180,E1 -14463.792,E2 -14463.792} C_VEL
LIN {X 0,Y 333.387,Z 418.806,A -85,B 0,C 180,E1 -14467.7,E2 -14467.7} C_VEL
LIN {X 0,Y 333.063,Z 425.596,A -85,B 0,C 180,E1 -14470.067,E2 -14470.067} C_VEL
LIN {X 0,Y 333.913,Z 440.603,A -85,B 0,C 180,E1 -14470.797,E2 -14470.797} C_VEL
LIN {X 0,Y 334.773,Z 454.323,A -85,B 0,C 180,E1 -14471.724,E2 -14471.724} C_VEL
LIN {X 0,Y 335.448,Z 466.517,A -85,B 0,C 180,E1 -14472.786,E2 -14472.786} C_VEL
LIN {X 0,Y 335.6,Z 475.492,A -85,B 0,C 180,E1 -14473.734,E2 -14473.734} C_VEL
LIN {X 0,Y 334.641,Z 485.822,A -85,B 0,C 180,E1 -14475.034,E2 -14475.034} C_VEL
LIN {X 0,Y 333.834,Z 495.949,A -85,B 0,C 180,E1 -14476.61,E2 -14476.61} C_VEL
LIN {X 0,Y 333.313,Z 503.999,A -85,B 0,C 180,E1 -14478.136,E2 -14478.136} C_VEL
LIN {X 0,Y 332.985,Z 511.931,A -85,B 0,C 180,E1 -14479.972,E2 -14479.972} C_VEL
LIN {X 0,Y 332.954,Z 517.306,A -85,B 0,C 180,E1 -14481.503,E2 -14481.503} C_VEL
LIN {X 0,Y 333.091,Z 522.957,A -85,B 0,C 180,E1 -14483.516,E2 -14483.516} C_VEL
LIN {X 0,Y 333.305,Z 526.454,A -85,B 0,C 180,E1 -14485.162,E2 -14485.162} C_VEL
LIN {X 0,Y 333.365,Z 528.399,A -85,B 0,C 180,E1 -14486.374,E2 -14486.374} C_VEL
LIN {X 0,Y 333.484,Z 529.872,A -85,B 0,C 180,E1 -14487.584,E2 -14487.584} C_VEL
LIN {X 0,Y 333.671,Z 530.91,A -85,B 0,C 180,E1 -14488.793,E2 -14488.793} C_VEL
LIN {X 0,Y 333.802,Z 531.476,A -85,B 0,C 180,E1 -14490,E2 -14490} C_VEL
LIN {X 0,Y 333.595,Z 531.512,A -85,B 0,C 180,E1 -14491.207,E2 -14491.207} C_VEL
LIN {X 0,Y 333.146,Z 530.289,A -85,B 0,C 180,E1 -14493.628,E2 -14493.628} C_VEL
LIN {X 0,Y 333.011,Z 529.03,A -85,B 0,C 180,E1 -14494.842,E2 -14494.842} C_VEL
LIN {X 0,Y 332.646,Z 525.136,A -85,B 0,C 180,E1 -14497.283,E2 -14497.283} C_VEL
LIN {X 0,Y 332.599,Z 521.045,A -85,B 0,C 180,E1 -14499.119,E2 -14499.119} C_VEL
LIN {X 0,Y 332.831,Z 515.9,A -85,B 0,C 180,E1 -14500.955,E2 -14500.955} C_VEL
LIN {X 0,Y 333.563,Z 508.452,A -85,B 0,C 180,E1 -14503.091,E2 -14503.091} C_VEL
LIN {X 0,Y 334.769,Z 499.447,A -85,B 0,C 180,E1 -14505.151,E2 -14505.151} C_VEL
LIN {X 0,Y 336.491,Z 489.525,A -85,B 0,C 180,E1 -14507.002,E2 -14507.002} C_VEL
LIN {X 0,Y 338.357,Z 478.935,A -85,B 0,C 180,E1 -14508.624,E2 -14508.624} C_VEL
LIN {X 0,Y 339.404,Z 467.565,A -85,B 0,C 180,E1 -14510.136,E2 -14510.136} C_VEL
LIN {X 0,Y 340.445,Z 455.223,A -85,B 0,C 180,E1 -14511.526,E2 -14511.526} C_VEL
LIN {X 0,Y 340.277,Z 443.048,A -85,B 0,C 180,E1 -14512.784,E2 -14512.784} C_VEL
LIN {X 0,Y 339.178,Z 431.524,A -85,B 0,C 180,E1 -14513.926,E2 -14513.926} C_VEL
LIN {X 0,Y 336.459,Z 416.697,A -85,B 0,C 180,E1 -14515.389,E2 -14515.389} C_VEL
LIN {X 0,Y 335.009,Z 411.047,A -85,B 0,C 180,E1 -14515.973,E2 -14515.973} C_VEL
LIN {X 0,Y 334.186,Z 406.936,A -85,B 0,C 180,E1 -14516.376,E2 -14516.376} C_VEL
LIN {X 0,Y 335.375,Z 394.983,A -85,B 0,C 180,E1 -14520.775,E2 -14520.775} C_VEL
LIN {X 0,Y 336.936,Z 384.471,A -85,B 0,C 180,E1 -14524.968,E2 -14524.968} C_VEL
LIN {X 0,Y 338.35,Z 377.774,A -85,B 0,C 180,E1 -14527.878,E2 -14527.878} C_VEL
LIN {X 0,Y 337.772,Z 373.412,A -85,B 0,C 180,E1 -14530.167,E2 -14530.167} C_VEL
LIN {X 0,Y 336.728,Z 367.907,A -85,B 0,C 180,E1 -14533.532,E2 -14533.532} C_VEL
LIN {X 0,Y 335.658,Z 363.135,A -85,B 0,C 180,E1 -14537.125,E2 -14537.125} C_VEL
LIN {X 0,Y 335.153,Z 360.567,A -85,B 0,C 180,E1 -14539.454,E2 -14539.454} C_VEL
LIN {X 0,Y 334.466,Z 357.502,A -85,B 0,C 180,E1 -14542.986,E2 -14542.986} C_VEL
LIN {X 0,Y 334.109,Z 355.934,A -85,B 0,C 180,E1 -14545.393,E2 -14545.393} C_VEL
LIN {X 0,Y 333.755,Z 354.569,A -85,B 0,C 180,E1 -14548.235,E2 -14548.235} C_VEL
LIN {X 0,Y 333.743,Z 353.91,A -85,B 0,C 180,E1 -14550.374,E2 -14550.374} C_VEL
LIN {X 0,Y 333.783,Z 354.003,A -85,B 0,C 180,E1 -14552.893,E2 -14552.893} C_VEL
LIN {X 0,Y 334.24,Z 355.709,A -85,B 0,C 180,E1 -14553.123,E2 -14553.123} C_VEL
LIN {X 0,Y 338.602,Z 362.832,A -85,B 0,C 180,E1 -14554.596,E2 -14554.596} C_VEL
LIN {X 0,Y 343.349,Z 372.999,A -85,B 0,C 180,E1 -14556.474,E2 -14556.474} C_VEL
LIN {X 0,Y 346.719,Z 382.498,A -85,B 0,C 180,E1 -14558.161,E2 -14558.161} C_VEL
LIN {X 0,Y 347.772,Z 387.214,A -85,B 0,C 180,E1 -14558.969,E2 -14558.969} C_VEL
LIN {X 0,Y 345.877,Z 397.902,A -85,B 0,C 180,E1 -14560.411,E2 -14560.411} C_VEL
LIN {X 0,Y 344.119,Z 406.608,A -85,B 0,C 180,E1 -14561.853,E2 -14561.853} C_VEL
LIN {X 0,Y 342.199,Z 415.111,A -85,B 0,C 180,E1 -14563.597,E2 -14563.597} C_VEL
LIN {X 0,Y 340.48,Z 422.07,A -85,B 0,C 180,E1 -14565.353,E2 -14565.353} C_VEL
LIN {X 0,Y 338.947,Z 427.96,A -85,B 0,C 180,E1 -14567.244,E2 -14567.244} C_VEL
LIN {X 0,Y 337.488,Z 432.604,A -85,B 0,C 180,E1 -14569.198,E2 -14569.198} C_VEL
LIN {X 0,Y 336.749,Z 434.826,A -85,B 0,C 180,E1 -14570.389,E2 -14570.389} C_VEL
LIN {X 0,Y 336.167,Z 436.609,A -85,B 0,C 180,E1 -14571.585,E2 -14571.585} C_VEL
LIN {X 0,Y 335.547,Z 437.953,A -85,B 0,C 180,E1 -14572.78,E2 -14572.78} C_VEL
LIN {X 0,Y 334.711,Z 439.395,A -85,B 0,C 180,E1 -14575.182,E2 -14575.182} C_VEL
LIN {X 0,Y 334.392,Z 439.526,A -85,B 0,C 180,E1 -14576.385,E2 -14576.385} C_VEL
LIN {X 0,Y 333.973,Z 438.536,A -85,B 0,C 180,E1 -14578.794,E2 -14578.794} C_VEL
LIN {X 0,Y 333.886,Z 437.455,A -85,B 0,C 180,E1 -14580,E2 -14580} C_VEL
LIN {X 0,Y 333.722,Z 435.954,A -85,B 0,C 180,E1 -14581.207,E2 -14581.207} C_VEL
LIN {X 0,Y 333.685,Z 432.897,A -85,B 0,C 180,E1 -14583.018,E2 -14583.018} C_VEL
LIN {X 0,Y 333.851,Z 428.808,A -85,B 0,C 180,E1 -14584.83,E2 -14584.83} C_VEL
LIN {X 0,Y 334.317,Z 423.582,A -85,B 0,C 180,E1 -14586.639,E2 -14586.639} C_VEL
LIN {X 0,Y 334.735,Z 417.115,A -85,B 0,C 180,E1 -14588.451,E2 -14588.451} C_VEL
LIN {X 0,Y 335.329,Z 409.195,A -85,B 0,C 180,E1 -14590.261,E2 -14590.261} C_VEL
LIN {X 0,Y 335.865,Z 401.202,A -85,B 0,C 180,E1 -14591.772,E2 -14591.772} C_VEL
LIN {X 0,Y 336.744,Z 390.478,A -85,B 0,C 180,E1 -14593.426,E2 -14593.426} C_VEL
LIN {X 0,Y 337.47,Z 379.783,A -85,B 0,C 180,E1 -14594.78,E2 -14594.78} C_VEL
LIN {X 0,Y 337.926,Z 371.214,A -85,B 0,C 180,E1 -14595.686,E2 -14595.686} C_VEL
LIN {X 0,Y 335.289,Z 360.204,A -85,B 0,C 180,E1 -14596.783,E2 -14596.783} C_VEL
LIN {X 0,Y 333.794,Z 353.908,A -85,B 0,C 180,E1 -14597.341,E2 -14597.341} C_VEL
LIN {X 0,Y 333.687,Z 353.921,A -85,B 0,C 180,E1 -14600.98,E2 -14600.98} C_VEL
LIN {X 0,Y 333.722,Z 353.918,A -85,B 0,C 180,E1 -14605.101,E2 -14605.101} C_VEL
LIN {X 0,Y 333.723,Z 353.912,A -85,B 0,C 180,E1 -14607.81,E2 -14607.81} C_VEL
LIN {X 0,Y 333.699,Z 353.916,A -85,B 0,C 180,E1 -14610.362,E2 -14610.362} C_VEL
LIN {X 0,Y 333.687,Z 353.921,A -85,B 0,C 180,E1 -14614.774,E2 -14614.774} C_VEL
LIN {X 0,Y 333.679,Z 353.923,A -85,B 0,C 180,E1 -14618.803,E2 -14618.803} C_VEL
LIN {X 0,Y 333.675,Z 353.921,A -85,B 0,C 180,E1 -14622.508,E2 -14622.508} C_VEL
LIN {X 0,Y 333.622,Z 353.925,A -85,B 0,C 180,E1 -14625.959,E2 -14625.959} C_VEL
LIN {X 0,Y 333.648,Z 353.922,A -85,B 0,C 180,E1 -14629.315,E2 -14629.315} C_VEL
LIN {X 0,Y 333.667,Z 353.92,A -85,B 0,C 180,E1 -14633.167,E2 -14633.167} C_VEL
LIN {X 0,Y 333.637,Z 353.926,A -85,B 0,C 180,E1 -14636.791,E2 -14636.791} C_VEL
LIN {X 0,Y 333.695,Z 353.916,A -85,B 0,C 180,E1 -14639.712,E2 -14639.712} C_VEL
LIN {X 0,Y 333.74,Z 353.915,A -85,B 0,C 180,E1 -14642.401,E2 -14642.401} C_VEL
LIN {X 0,Y 333.728,Z 353.912,A -85,B 0,C 180,E1 -14645.091,E2 -14645.091} C_VEL
LIN {X 0,Y 333.694,Z 353.916,A -85,B 0,C 180,E1 -14649.02,E2 -14649.02} C_VEL
LIN {X 0,Y 333.796,Z 353.903,A -85,B 0,C 180,E1 -14651.589,E2 -14651.589} C_VEL
LIN {X 0,Y 333.809,Z 353.902,A -85,B 0,C 180,E1 -14655.577,E2 -14655.577} C_VEL
LIN {X 0,Y 333.835,Z 353.898,A -85,B 0,C 180,E1 -14659.078,E2 -14659.078} C_VEL
LIN {X 0,Y 334.006,Z 353.878,A -85,B 0,C 180,E1 -14662.747,E2 -14662.747} C_VEL
LIN {X 0,Y 333.81,Z 353.901,A -85,B 0,C 180,E1 -14665.169,E2 -14665.169} C_VEL
LIN {X 0,Y 334.108,Z 353.866,A -85,B 0,C 180,E1 -14667.589,E2 -14667.589} C_VEL
LIN {X 0,Y 334.247,Z 353.853,A -85,B 0,C 180,E1 -14670,E2 -14670} C_VEL
LIN {X 0,Y 334.109,Z 353.866,A -85,B 0,C 180,E1 -14672.411,E2 -14672.411} C_VEL
LIN {X 0,Y 334.015,Z 353.88,A -85,B 0,C 180,E1 -14676.039,E2 -14676.039} C_VEL
LIN {X 0,Y 333.959,Z 353.884,A -85,B 0,C 180,E1 -14678.471,E2 -14678.471} C_VEL
LIN {X 0,Y 333.792,Z 353.906,A -85,B 0,C 180,E1 -14682.155,E2 -14682.155} C_VEL
LIN {X 0,Y 333.779,Z 353.909,A -85,B 0,C 180,E1 -14685.886,E2 -14685.886} C_VEL
LIN {X 0,Y 333.798,Z 353.903,A -85,B 0,C 180,E1 -14688.656,E2 -14688.656} C_VEL
LIN {X 0,Y 333.693,Z 353.917,A -85,B 0,C 180,E1 -14692.278,E2 -14692.278} C_VEL
LIN {X 0,Y 333.736,Z 353.911,A -85,B 0,C 180,E1 -14696.247,E2 -14696.247} C_VEL
LIN {X 0,Y 333.691,Z 353.917,A -85,B 0,C 180,E1 -14698.974,E2 -14698.974} C_VEL
LIN {X 0,Y 333.644,Z 353.922,A -85,B 0,C 180,E1 -14702.587,E2 -14702.587} C_VEL
LIN {X 0,Y 333.677,Z 353.918,A -85,B 0,C 180,E1 -14706.139,E2 -14706.139} C_VEL
LIN {X 0,Y 333.683,Z 353.921,A -85,B 0,C 180,E1 -14709.188,E2 -14709.188} C_VEL
LIN {X 0,Y 333.691,Z 353.916,A -85,B 0,C 180,E1 -14712.511,E2 -14712.511} C_VEL
LIN {X 0,Y 333.636,Z 353.923,A -85,B 0,C 180,E1 -14715.962,E2 -14715.962} C_VEL
LIN {X 0,Y 333.649,Z 353.926,A -85,B 0,C 180,E1 -14719.316,E2 -14719.316} C_VEL
LIN {X 0,Y 333.667,Z 353.924,A -85,B 0,C 180,E1 -14723.168,E2 -14723.168} C_VEL
LIN {X 0,Y 333.677,Z 353.921,A -85,B 0,C 180,E1 -14725.342,E2 -14725.342} C_VEL
LIN {X 0,Y 333.705,Z 353.915,A -85,B 0,C 180,E1 -14729.711,E2 -14729.711} C_VEL
LIN {X 0,Y 333.746,Z 353.91,A -85,B 0,C 180,E1 -14732.402,E2 -14732.402} C_VEL
LIN {X 0,Y 333.731,Z 353.915,A -85,B 0,C 180,E1 -14735.091,E2 -14735.091} C_VEL
LIN {X 0,Y 333.674,Z 353.916,A -85,B 0,C 180,E1 -14737.384,E2 -14737.384} C_VEL
LIN {X 0,Y 333.052,Z 353.999,A -85,B 0,C 180,E1 -14738.391,E2 -14738.391} C_VEL
LIN {X 0,Y 330.236,Z 354.354,A -85,B 0,C 180,E1 -14740.031,E2 -14740.031} C_VEL
LIN {X 0,Y 327.823,Z 354.654,A -85,B 0,C 180,E1 -14741.36,E2 -14741.36} C_VEL
LIN {X 0,Y 326.782,Z 354.779,A -85,B 0,C 180,E1 -14742.388,E2 -14742.388} C_VEL
LIN {X 0,Y 326.696,Z 354.788,A -85,B 0,C 180,E1 -14742.736,E2 -14742.736} C_VEL
LIN {X 0,Y 326.763,Z 354.781,A -85,B 0,C 180,E1 -14746.315,E2 -14746.315} C_VEL
LIN {X 0,Y 326.818,Z 354.773,A -85,B 0,C 180,E1 -14750.094,E2 -14750.094} C_VEL
LIN {X 0,Y 326.984,Z 354.757,A -85,B 0,C 180,E1 -14752.591,E2 -14752.591} C_VEL
LIN {X 0,Y 326.78,Z 354.778,A -85,B 0,C 180,E1 -14755.065,E2 -14755.065} C_VEL
LIN {X 0,Y 327.05,Z 354.743,A -85,B 0,C 180,E1 -14757.537,E2 -14757.537} C_VEL
LIN {X 0,Y 327.202,Z 354.726,A -85,B 0,C 180,E1 -14760,E2 -14760} C_VEL
LIN {X 0,Y 327.052,Z 354.749,A -85,B 0,C 180,E1 -14762.463,E2 -14762.463} C_VEL
LIN {X 0,Y 326.987,Z 354.755,A -85,B 0,C 180,E1 -14766.169,E2 -14766.169} C_VEL
LIN {X 0,Y 326.809,Z 354.775,A -85,B 0,C 180,E1 -14769.907,E2 -14769.907} C_VEL
LIN {X 0,Y 326.764,Z 354.78,A -85,B 0,C 180,E1 -14773.685,E2 -14773.685} C_VEL
LIN {X 0,Y 326.704,Z 354.787,A -85,B 0,C 180,E1 -14777.528,E2 -14777.528} C_VEL
LIN {X 0,Y 326.669,Z 354.796,A -85,B 0,C 180,E1 -14780.135,E2 -14780.135} C_VEL
LIN {X 0,Y 326.656,Z 354.798,A -85,B 0,C 180,E1 -14784.129,E2 -14784.129} C_VEL
LIN {X 0,Y 326.689,Z 354.788,A -85,B 0,C 180,E1 -14786.858,E2 -14786.858} C_VEL
LIN {X 0,Y 326.643,Z 354.795,A -85,B 0,C 180,E1 -14790.611,E2 -14790.611} C_VEL
LIN {X 0,Y 326.612,Z 354.803,A -85,B 0,C 180,E1 -14794.019,E2 -14794.019} C_VEL
LIN {X 0,Y 326.632,Z 354.796,A -85,B 0,C 180,E1 -14797.239,E2 -14797.239} C_VEL
LIN {X 0,Y 326.584,Z 354.802,A -85,B 0,C 180,E1 -14801.132,E2 -14801.132} C_VEL
LIN {X 0,Y 326.67,Z 354.996,A -85,B 0,C 180,E1 -14803.348,E2 -14803.348} C_VEL
LIN {X 0,Y 328.172,Z 362.902,A -85,B 0,C 180,E1 -14806.74,E2 -14806.74} C_VEL
LIN {X 0,Y 330.117,Z 372.535,A -85,B 0,C 180,E1 -14810.701,E2 -14810.701} C_VEL
LIN {X 0,Y 330.67,Z 375.685,A -85,B 0,C 180,E1 -14811.949,E2 -14811.949} C_VEL
LIN {X 0,Y 330.162,Z 381.099,A -85,B 0,C 180,E1 -14813.988,E2 -14813.988} C_VEL
LIN {X 0,Y 328.862,Z 391.163,A -85,B 0,C 180,E1 -14817.705,E2 -14817.705} C_VEL
LIN {X 0,Y 327.628,Z 402.522,A -85,B 0,C 180,E1 -14821.84,E2 -14821.84} C_VEL
LIN {X 0,Y 326.64,Z 413.7,A -85,B 0,C 180,E1 -14825.87,E2 -14825.87} C_VEL
LIN {X 0,Y 326,Z 424.711,A -85,B 0,C 180,E1 -14829.822,E2 -14829.822} C_VEL
LIN {X 0,Y 326.834,Z 439.951,A -85,B 0,C 180,E1 -14830.585,E2 -14830.585} C_VEL
LIN {X 0,Y 327.671,Z 453.856,A -85,B 0,C 180,E1 -14831.557,E2 -14831.557} C_VEL
LIN {X 0,Y 328.363,Z 466.773,A -85,B 0,C 180,E1 -14832.724,E2 -14832.724} C_VEL
LIN {X 0,Y 328.509,Z 475.531,A -85,B 0,C 180,E1 -14833.692,E2 -14833.692} C_VEL
LIN {X 0,Y 327.51,Z 486.02,A -85,B 0,C 180,E1 -14835.078,E2 -14835.078} C_VEL
LIN {X 0,Y 326.768,Z 495.586,A -85,B 0,C 180,E1 -14836.632,E2 -14836.632} C_VEL
LIN {X 0,Y 326.255,Z 503.515,A -85,B 0,C 180,E1 -14838.191,E2 -14838.191} C_VEL
LIN {X 0,Y 325.928,Z 511.328,A -85,B 0,C 180,E1 -14840.066,E2 -14840.066} C_VEL
LIN {X 0,Y 325.934,Z 517.554,A -85,B 0,C 180,E1 -14841.943,E2 -14841.943} C_VEL
LIN {X 0,Y 326.11,Z 522.432,A -85,B 0,C 180,E1 -14843.814,E2 -14843.814} C_VEL
LIN {X 0,Y 326.314,Z 526.077,A -85,B 0,C 180,E1 -14845.677,E2 -14845.677} C_VEL
LIN {X 0,Y 326.482,Z 528.578,A -85,B 0,C 180,E1 -14847.532,E2 -14847.532} C_VEL
LIN {X 0,Y 326.664,Z 529.657,A -85,B 0,C 180,E1 -14848.767,E2 -14848.767} C_VEL
LIN {X 0,Y 326.819,Z 530.29,A -85,B 0,C 180,E1 -14850,E2 -14850} C_VEL
LIN {X 0,Y 326.586,Z 530.392,A -85,B 0,C 180,E1 -14851.233,E2 -14851.233} C_VEL
LIN {X 0,Y 326.095,Z 529.247,A -85,B 0,C 180,E1 -14853.707,E2 -14853.707} C_VEL
LIN {X 0,Y 325.944,Z 528.05,A -85,B 0,C 180,E1 -14854.948,E2 -14854.948} C_VEL
LIN {X 0,Y 325.625,Z 525.306,A -85,B 0,C 180,E1 -14856.867,E2 -14856.867} C_VEL
LIN {X 0,Y 325.504,Z 521.743,A -85,B 0,C 180,E1 -14858.693,E2 -14858.693} C_VEL
LIN {X 0,Y 325.661,Z 517.073,A -85,B 0,C 180,E1 -14860.57,E2 -14860.57} C_VEL
LIN {X 0,Y 326.371,Z 510.27,A -85,B 0,C 180,E1 -14862.751,E2 -14862.751} C_VEL
LIN {X 0,Y 327.438,Z 501.747,A -85,B 0,C 180,E1 -14864.926,E2 -14864.926} C_VEL
LIN {X 0,Y 329.068,Z 492.924,A -85,B 0,C 180,E1 -14866.758,E2 -14866.758} C_VEL
LIN {X 0,Y 331.141,Z 482.35,A -85,B 0,C 180,E1 -14868.563,E2 -14868.563} C_VEL
LIN {X 0,Y 332.683,Z 469.652,A -85,B 0,C 180,E1 -14870.4,E2 -14870.4} C_VEL
LIN {X 0,Y 333.934,Z 457.458,A -85,B 0,C 180,E1 -14871.877,E2 -14871.877} C_VEL
LIN {X 0,Y 334.085,Z 445.249,A -85,B 0,C 180,E1 -14873.231,E2 -14873.231} C_VEL
LIN {X 0,Y 333.042,Z 432.769,A -85,B 0,C 180,E1 -14874.572,E2 -14874.572} C_VEL
LIN {X 0,Y 330.971,Z 419.695,A -85,B 0,C 180,E1 -14875.962,E2 -14875.962} C_VEL
LIN {X 0,Y 328.62,Z 409.818,A -85,B 0,C 180,E1 -14877.065,E2 -14877.065} C_VEL
LIN {X 0,Y 327.455,Z 405.173,A -85,B 0,C 180,E1 -14877.589,E2 -14877.589} C_VEL
LIN {X 0,Y 327.483,Z 404.213,A -85,B 0,C 180,E1 -14877.825,E2 -14877.825} C_VEL
LIN {X 0,Y 328.636,Z 394.276,A -85,B 0,C 180,E1 -14881.653,E2 -14881.653} C_VEL
LIN {X 0,Y 330.255,Z 384.783,A -85,B 0,C 180,E1 -14885.597,E2 -14885.597} C_VEL
LIN {X 0,Y 331.446,Z 379.534,A -85,B 0,C 180,E1 -14887.946,E2 -14887.946} C_VEL
LIN {X 0,Y 330.973,Z 375.431,A -85,B 0,C 180,E1 -14890.143,E2 -14890.143} C_VEL
LIN {X 0,Y 329.925,Z 369.912,A -85,B 0,C 180,E1 -14893.592,E2 -14893.592} C_VEL
LIN {X 0,Y 328.949,Z 365.602,A -85,B 0,C 180,E1 -14896.868,E2 -14896.868} C_VEL
LIN {X 0,Y 328.245,Z 362.206,A -85,B 0,C 180,E1 -14900.034,E2 -14900.034} C_VEL
LIN {X 0,Y 327.7,Z 359.637,A -85,B 0,C 180,E1 -14903.094,E2 -14903.094} C_VEL
LIN {X 0,Y 327.189,Z 357.33,A -85,B 0,C 180,E1 -14906.9,E2 -14906.9} C_VEL
LIN {X 0,Y 326.883,Z 355.806,A -85,B 0,C 180,E1 -14911.07,E2 -14911.07} C_VEL
LIN {X 0,Y 326.86,Z 355.811,A -85,B 0,C 180,E1 -14911.539,E2 -14911.539} C_VEL
LIN {X 0,Y 327.532,Z 357.389,A -85,B 0,C 180,E1 -14911.831,E2 -14911.831} C_VEL
LIN {X 0,Y 329.153,Z 359.326,A -85,B 0,C 180,E1 -14912.387,E2 -14912.387} C_VEL
LIN {X 0,Y 334.092,Z 368.184,A -85,B 0,C 180,E1 -14914.307,E2 -14914.307} C_VEL
LIN {X 0,Y 338.164,Z 377.346,A -85,B 0,C 180,E1 -14916.128,E2 -14916.128} C_VEL
LIN {X 0,Y 341.23,Z 386.921,A -85,B 0,C 180,E1 -14917.946,E2 -14917.946} C_VEL
LIN {X 0,Y 341.64,Z 388.654,A -85,B 0,C 180,E1 -14918.267,E2 -14918.267} C_VEL
LIN {X 0,Y 341.5,Z 391.389,A -85,B 0,C 180,E1 -14918.675,E2 -14918.675} C_VEL
LIN {X 0,Y 339.618,Z 400.84,A -85,B 0,C 180,E1 -14920.035,E2 -14920.035} C_VEL
LIN {X 0,Y 337.437,Z 410.706,A -85,B 0,C 180,E1 -14921.795,E2 -14921.795} C_VEL
LIN {X 0,Y 335.392,Z 418.714,A -85,B 0,C 180,E1 -14923.567,E2 -14923.567} C_VEL
LIN {X 0,Y 333.308,Z 426.147,A -85,B 0,C 180,E1 -14925.686,E2 -14925.686} C_VEL
LIN {X 0,Y 331.658,Z 431.755,A -85,B 0,C 180,E1 -14927.766,E2 -14927.766} C_VEL
LIN {X 0,Y 330.387,Z 435.432,A -85,B 0,C 180,E1 -14929.583,E2 -14929.583} C_VEL
LIN {X 0,Y 329.313,Z 438.103,A -85,B 0,C 180,E1 -14931.408,E2 -14931.408} C_VEL
LIN {X 0,Y 328.158,Z 440.206,A -85,B 0,C 180,E1 -14933.853,E2 -14933.853} C_VEL
LIN {X 0,Y 327.75,Z 440.667,A -85,B 0,C 180,E1 -14935.079,E2 -14935.079} C_VEL
LIN {X 0,Y 327.137,Z 440.328,A -85,B 0,C 180,E1 -14937.537,E2 -14937.537} C_VEL
LIN {X 0,Y 326.953,Z 439.568,A -85,B 0,C 180,E1 -14938.768,E2 -14938.768} C_VEL
LIN {X 0,Y 326.862,Z 438.398,A -85,B 0,C 180,E1 -14940,E2 -14940} C_VEL
LIN {X 0,Y 326.728,Z 435.877,A -85,B 0,C 180,E1 -14941.849,E2 -14941.849} C_VEL
LIN {X 0,Y 326.543,Z 432.383,A -85,B 0,C 180,E1 -14943.702,E2 -14943.702} C_VEL
LIN {X 0,Y 327.074,Z 427.768,A -85,B 0,C 180,E1 -14945.549,E2 -14945.549} C_VEL
LIN {X 0,Y 327.474,Z 420.911,A -85,B 0,C 180,E1 -14947.708,E2 -14947.708} C_VEL
LIN {X 0,Y 328.09,Z 412.44,A -85,B 0,C 180,E1 -14949.813,E2 -14949.813} C_VEL
LIN {X 0,Y 328.761,Z 402.866,A -85,B 0,C 180,E1 -14951.717,E2 -14951.717} C_VEL
LIN {X 0,Y 329.647,Z 392.349,A -85,B 0,C 180,E1 -14953.406,E2 -14953.406} C_VEL
LIN {X 0,Y 330.469,Z 380.583,A -85,B 0,C 180,E1 -14954.943,E2 -14954.943} C_VEL
LIN {X 0,Y 330.911,Z 372.012,A -85,B 0,C 180,E1 -14955.869,E2 -14955.869} C_VEL
LIN {X 0,Y 328.166,Z 360.756,A -85,B 0,C 180,E1 -14957.005,E2 -14957.005} C_VEL
LIN {X 0,Y 326.725,Z 354.786,A -85,B 0,C 180,E1 -14957.526,E2 -14957.526} C_VEL
LIN {X 0,Y 326.651,Z 354.796,A -85,B 0,C 180,E1 -14961.454,E2 -14961.454} C_VEL
LIN {X 0,Y 326.692,Z 354.79,A -85,B 0,C 180,E1 -14965.483,E2 -14965.483} C_VEL
LIN {X 0,Y 326.662,Z 354.792,A -85,B 0,C 180,E1 -14969.659,E2 -14969.659} C_VEL
LIN {X 0,Y 326.609,Z 354.798,A -85,B 0,C 180,E1 -14974.019,E2 -14974.019} C_VEL
LIN {X 0,Y 326.631,Z 354.798,A -85,B 0,C 180,E1 -14977.239,E2 -14977.239} C_VEL
LIN {X 0,Y 326.605,Z 354.799,A -85,B 0,C 180,E1 -14980.207,E2 -14980.207} C_VEL
LIN {X 0,Y 326.602,Z 354.799,A -85,B 0,C 180,E1 -14983.519,E2 -14983.519} C_VEL
LIN {X 0,Y 326.583,Z 354.804,A -85,B 0,C 180,E1 -14987.027,E2 -14987.027} C_VEL
LIN {X 0,Y 326.613,Z 354.802,A -85,B 0,C 180,E1 -14990.772,E2 -14990.772} C_VEL
LIN {X 0,Y 326.614,Z 354.802,A -85,B 0,C 180,E1 -14994.48,E2 -14994.48} C_VEL
LIN {X 0,Y 326.608,Z 354.798,A -85,B 0,C 180,E1 -14997.455,E2 -14997.455} C_VEL
LIN {X 0,Y 326.648,Z 354.797,A -85,B 0,C 180,E1 -15000.34,E2 -15000.34} C_VEL
LIN {X 0,Y 326.69,Z 354.793,A -85,B 0,C 180,E1 -15004.516,E2 -15004.516} C_VEL
LIN {X 0,Y 326.653,Z 354.796,A -85,B 0,C 180,E1 -15008.546,E2 -15008.546} C_VEL
LIN {X 0,Y 326.745,Z 354.781,A -85,B 0,C 180,E1 -15011.177,E2 -15011.177} C_VEL
LIN {X 0,Y 326.764,Z 354.779,A -85,B 0,C 180,E1 -15015.433,E2 -15015.433} C_VEL
LIN {X 0,Y 326.771,Z 354.779,A -85,B 0,C 180,E1 -15018.839,E2 -15018.839} C_VEL
LIN {X 0,Y 326.958,Z 354.756,A -85,B 0,C 180,E1 -15022.59,E2 -15022.59} C_VEL
LIN {X 0,Y 326.777,Z 354.777,A -85,B 0,C 180,E1 -15025.065,E2 -15025.065} C_VEL
LIN {X 0,Y 327.049,Z 354.745,A -85,B 0,C 180,E1 -15027.537,E2 -15027.537} C_VEL
LIN {X 0,Y 327.198,Z 354.731,A -85,B 0,C 180,E1 -15030,E2 -15030} C_VEL
LIN {X 0,Y 327.049,Z 354.745,A -85,B 0,C 180,E1 -15032.463,E2 -15032.463} C_VEL
LIN {X 0,Y 326.99,Z 354.754,A -85,B 0,C 180,E1 -15036.169,E2 -15036.169} C_VEL
LIN {X 0,Y 326.807,Z 354.779,A -85,B 0,C 180,E1 -15039.907,E2 -15039.907} C_VEL
LIN {X 0,Y 326.76,Z 354.784,A -85,B 0,C 180,E1 -15043.686,E2 -15043.686} C_VEL
LIN {X 0,Y 326.701,Z 354.791,A -85,B 0,C 180,E1 -15047.528,E2 -15047.528} C_VEL
LIN {X 0,Y 326.666,Z 354.793,A -85,B 0,C 180,E1 -15050.135,E2 -15050.135} C_VEL
LIN {X 0,Y 326.654,Z 354.794,A -85,B 0,C 180,E1 -15054.129,E2 -15054.129} C_VEL
LIN {X 0,Y 326.684,Z 354.789,A -85,B 0,C 180,E1 -15056.858,E2 -15056.858} C_VEL
LIN {X 0,Y 326.635,Z 354.795,A -85,B 0,C 180,E1 -15060.61,E2 -15060.61} C_VEL
LIN {X 0,Y 326.608,Z 354.799,A -85,B 0,C 180,E1 -15064.02,E2 -15064.02} C_VEL
LIN {X 0,Y 326.629,Z 354.8,A -85,B 0,C 180,E1 -15067.239,E2 -15067.239} C_VEL
LIN {X 0,Y 326.636,Z 354.795,A -85,B 0,C 180,E1 -15070.203,E2 -15070.203} C_VEL
LIN {X 0,Y 326.621,Z 354.8,A -85,B 0,C 180,E1 -15073.516,E2 -15073.516} C_VEL
LIN {X 0,Y 326.588,Z 354.805,A -85,B 0,C 180,E1 -15077.027,E2 -15077.027} C_VEL
LIN {X 0,Y 326.613,Z 354.8,A -85,B 0,C 180,E1 -15080.773,E2 -15080.773} C_VEL
LIN {X 0,Y 326.615,Z 354.798,A -85,B 0,C 180,E1 -15084.481,E2 -15084.481} C_VEL
LIN {X 0,Y 326.61,Z 354.8,A -85,B 0,C 180,E1 -15087.456,E2 -15087.456} C_VEL
LIN {X 0,Y 326.663,Z 354.792,A -85,B 0,C 180,E1 -15090.341,E2 -15090.341} C_VEL
LIN {X 0,Y 326.693,Z 354.79,A -85,B 0,C 180,E1 -15094.517,E2 -15094.517} C_VEL
LIN {X 0,Y 326.652,Z 354.796,A -85,B 0,C 180,E1 -15098.546,E2 -15098.546} C_VEL
LIN {X 0,Y 326.748,Z 354.783,A -85,B 0,C 180,E1 -15101.178,E2 -15101.178} C_VEL
LIN {X 0,Y 326.696,Z 354.788,A -85,B 0,C 180,E1 -15102.736,E2 -15102.736} C_VEL
LIN {X 0,Y 326.019,Z 354.872,A -85,B 0,C 180,E1 -15103.766,E2 -15103.766} C_VEL
LIN {X 0,Y 323.155,Z 355.229,A -85,B 0,C 180,E1 -15105.442,E2 -15105.442} C_VEL
LIN {X 0,Y 320.756,Z 355.532,A -85,B 0,C 180,E1 -15106.8,E2 -15106.8} C_VEL
LIN {X 0,Y 319.761,Z 355.652,A -85,B 0,C 180,E1 -15107.851,E2 -15107.851} C_VEL
LIN {X 0,Y 319.698,Z 355.66,A -85,B 0,C 180,E1 -15108.207,E2 -15108.207} C_VEL
LIN {X 0,Y 319.938,Z 355.633,A -85,B 0,C 180,E1 -15112.427,E2 -15112.427} C_VEL
LIN {X 0,Y 319.75,Z 355.655,A -85,B 0,C 180,E1 -15114.956,E2 -15114.956} C_VEL
LIN {X 0,Y 319.994,Z 355.622,A -85,B 0,C 180,E1 -15117.483,E2 -15117.483} C_VEL
LIN {X 0,Y 320.154,Z 355.603,A -85,B 0,C 180,E1 -15120,E2 -15120} C_VEL
LIN {X 0,Y 319.996,Z 355.627,A -85,B 0,C 180,E1 -15122.518,E2 -15122.518} C_VEL
LIN {X 0,Y 319.94,Z 355.634,A -85,B 0,C 180,E1 -15126.306,E2 -15126.306} C_VEL
LIN {X 0,Y 319.756,Z 355.655,A -85,B 0,C 180,E1 -15130.127,E2 -15130.127} C_VEL
LIN {X 0,Y 319.735,Z 355.656,A -85,B 0,C 180,E1 -15134.724,E2 -15134.724} C_VEL
LIN {X 0,Y 319.694,Z 355.66,A -85,B 0,C 180,E1 -15139.038,E2 -15139.038} C_VEL
LIN {X 0,Y 319.575,Z 355.675,A -85,B 0,C 180,E1 -15143.319,E2 -15143.319} C_VEL
LIN {X 0,Y 319.639,Z 355.672,A -85,B 0,C 180,E1 -15146.088,E2 -15146.088} C_VEL
LIN {X 0,Y 319.593,Z 355.672,A -85,B 0,C 180,E1 -15148.934,E2 -15148.934} C_VEL
LIN {X 0,Y 319.537,Z 355.684,A -85,B 0,C 180,E1 -15151.861,E2 -15151.861} C_VEL
LIN {X 0,Y 319.584,Z 355.675,A -85,B 0,C 180,E1 -15155.543,E2 -15155.543} C_VEL
LIN {X 0,Y 319.577,Z 355.678,A -85,B 0,C 180,E1 -15158.008,E2 -15158.008} C_VEL
LIN {X 0,Y 319.561,Z 355.68,A -85,B 0,C 180,E1 -15161.603,E2 -15161.603} C_VEL
LIN {X 0,Y 319.609,Z 355.842,A -85,B 0,C 180,E1 -15163.077,E2 -15163.077} C_VEL
LIN {X 0,Y 321.22,Z 364.318,A -85,B 0,C 180,E1 -15166.8,E2 -15166.8} C_VEL
LIN {X 0,Y 323.209,Z 374.123,A -85,B 0,C 180,E1 -15170.906,E2 -15170.906} C_VEL
LIN {X 0,Y 323.606,Z 378.229,A -85,B 0,C 180,E1 -15172.548,E2 -15172.548} C_VEL
LIN {X 0,Y 322.193,Z 388.459,A -85,B 0,C 180,E1 -15176.433,E2 -15176.433} C_VEL
LIN {X 0,Y 320.883,Z 399.239,A -85,B 0,C 180,E1 -15180.475,E2 -15180.475} C_VEL
LIN {X 0,Y 319.807,Z 410.84,A -85,B 0,C 180,E1 -15184.782,E2 -15184.782} C_VEL
LIN {X 0,Y 319.034,Z 421.403,A -85,B 0,C 180,E1 -15188.686,E2 -15188.686} C_VEL
LIN {X 0,Y 318.928,Z 423.807,A -85,B 0,C 180,E1 -15189.565,E2 -15189.565} C_VEL
LIN {X 0,Y 319.775,Z 440.02,A -85,B 0,C 180,E1 -15190.417,E2 -15190.417} C_VEL
LIN {X 0,Y 320.627,Z 454.256,A -85,B 0,C 180,E1 -15191.468,E2 -15191.468} C_VEL
LIN {X 0,Y 321.283,Z 466.797,A -85,B 0,C 180,E1 -15192.66,E2 -15192.66} C_VEL
LIN {X 0,Y 321.403,Z 475.547,A -85,B 0,C 180,E1 -15193.664,E2 -15193.664} C_VEL
LIN {X 0,Y 320.385,Z 486.484,A -85,B 0,C 180,E1 -15195.186,E2 -15195.186} C_VEL
LIN {X 0,Y 319.633,Z 496.876,A -85,B 0,C 180,E1 -15196.975,E2 -15196.975} C_VEL
LIN {X 0,Y 319.086,Z 505.722,A -85,B 0,C 180,E1 -15198.888,E2 -15198.888} C_VEL
LIN {X 0,Y 318.916,Z 512.879,A -85,B 0,C 180,E1 -15200.806,E2 -15200.806} C_VEL
LIN {X 0,Y 319.014,Z 519.044,A -85,B 0,C 180,E1 -15202.915,E2 -15202.915} C_VEL
LIN {X 0,Y 319.262,Z 523.524,A -85,B 0,C 180,E1 -15204.948,E2 -15204.948} C_VEL
LIN {X 0,Y 319.348,Z 525.634,A -85,B 0,C 180,E1 -15206.214,E2 -15206.214} C_VEL
LIN {X 0,Y 319.478,Z 527.26,A -85,B 0,C 180,E1 -15207.478,E2 -15207.478} C_VEL
LIN {X 0,Y 319.656,Z 528.388,A -85,B 0,C 180,E1 -15208.74,E2 -15208.74} C_VEL
LIN {X 0,Y 319.83,Z 529.07,A -85,B 0,C 180,E1 -15210,E2 -15210} C_VEL
LIN {X 0,Y 319.572,Z 529.243,A -85,B 0,C 180,E1 -15211.26,E2 -15211.26} C_VEL
LIN {X 0,Y 319.193,Z 528.933,A -85,B 0,C 180,E1 -15212.524,E2 -15212.524} C_VEL
LIN {X 0,Y 319.044,Z 528.206,A -85,B 0,C 180,E1 -15213.789,E2 -15213.789} C_VEL
LIN {X 0,Y 318.878,Z 527.056,A -85,B 0,C 180,E1 -15215.058,E2 -15215.058} C_VEL
LIN {X 0,Y 318.556,Z 524.634,A -85,B 0,C 180,E1 -15216.882,E2 -15216.882} C_VEL
LIN {X 0,Y 318.42,Z 520.966,A -85,B 0,C 180,E1 -15218.888,E2 -15218.888} C_VEL
LIN {X 0,Y 318.767,Z 514.708,A -85,B 0,C 180,E1 -15221.445,E2 -15221.445} C_VEL
LIN {X 0,Y 319.641,Z 507.6,A -85,B 0,C 180,E1 -15223.672,E2 -15223.672} C_VEL
LIN {X 0,Y 320.8,Z 500.333,A -85,B 0,C 180,E1 -15225.534,E2 -15225.534} C_VEL
LIN {X 0,Y 322.587,Z 491.38,A -85,B 0,C 180,E1 -15227.431,E2 -15227.431} C_VEL
LIN {X 0,Y 324.78,Z 480.85,A -85,B 0,C 180,E1 -15229.269,E2 -15229.269} C_VEL
LIN {X 0,Y 326.259,Z 469.4,A -85,B 0,C 180,E1 -15230.985,E2 -15230.985} C_VEL
LIN {X 0,Y 327.622,Z 457.749,A -85,B 0,C 180,E1 -15232.473,E2 -15232.473} C_VEL
LIN {X 0,Y 327.875,Z 446.018,A -85,B 0,C 180,E1 -15233.865,E2 -15233.865} C_VEL
LIN {X 0,Y 327.037,Z 434.168,A -85,B 0,C 180,E1 -15235.234,E2 -15235.234} C_VEL
LIN {X 0,Y 325.031,Z 420.432,A -85,B 0,C 180,E1 -15236.814,E2 -15236.814} C_VEL
LIN {X 0,Y 322.112,Z 407.796,A -85,B 0,C 180,E1 -15238.371,E2 -15238.371} C_VEL
LIN {X 0,Y 320.893,Z 403.213,A -85,B 0,C 180,E1 -15238.966,E2 -15238.966} C_VEL
LIN {X 0,Y 320.854,Z 402.159,A -85,B 0,C 180,E1 -15239.131,E2 -15239.131} C_VEL
LIN {X 0,Y 322.187,Z 392.482,A -85,B 0,C 180,E1 -15243.048,E2 -15243.048} C_VEL
LIN {X 0,Y 324.242,Z 382.679,A -85,B 0,C 180,E1 -15247.366,E2 -15247.366} C_VEL
LIN {X 0,Y 324.552,Z 381.234,A -85,B 0,C 180,E1 -15248.047,E2 -15248.047} C_VEL
LIN {X 0,Y 324.267,Z 378.105,A -85,B 0,C 180,E1 -15249.745,E2 -15249.745} C_VEL
LIN {X 0,Y 323.265,Z 372.485,A -85,B 0,C 180,E1 -15253.254,E2 -15253.254} C_VEL
LIN {X 0,Y 322.433,Z 368.823,A -85,B 0,C 180,E1 -15255.997,E2 -15255.997} C_VEL
LIN {X 0,Y 321.522,Z 364.531,A -85,B 0,C 180,E1 -15259.912,E2 -15259.912} C_VEL
LIN {X 0,Y 321.113,Z 362.532,A -85,B 0,C 180,E1 -15262.206,E2 -15262.206} C_VEL
LIN {X 0,Y 320.61,Z 360.444,A -85,B 0,C 180,E1 -15265.254,E2 -15265.254} C_VEL
LIN {X 0,Y 320.236,Z 358.707,A -85,B 0,C 180,E1 -15268.861,E2 -15268.861} C_VEL
LIN {X 0,Y 320.246,Z 358.4,A -85,B 0,C 180,E1 -15270.11,E2 -15270.11} C_VEL
LIN {X 0,Y 321.956,Z 360.924,A -85,B 0,C 180,E1 -15270.829,E2 -15270.829} C_VEL
LIN {X 0,Y 324.514,Z 364.049,A -85,B 0,C 180,E1 -15271.802,E2 -15271.802} C_VEL
LIN {X 0,Y 329.032,Z 372.374,A -85,B 0,C 180,E1 -15273.781,E2 -15273.781} C_VEL
LIN {X 0,Y 332.305,Z 380.026,A -85,B 0,C 180,E1 -15275.426,E2 -15275.426} C_VEL
LIN {X 0,Y 335.223,Z 389.13,A -85,B 0,C 180,E1 -15277.29,E2 -15277.29} C_VEL
LIN {X 0,Y 335.819,Z 392.066,A -85,B 0,C 180,E1 -15277.87,E2 -15277.87} C_VEL
LIN {X 0,Y 333.828,Z 402.059,A -85,B 0,C 180,E1 -15279.351,E2 -15279.351} C_VEL
LIN {X 0,Y 331.455,Z 411.851,A -85,B 0,C 180,E1 -15281.134,E2 -15281.134} C_VEL
LIN {X 0,Y 329.292,Z 419.842,A -85,B 0,C 180,E1 -15282.934,E2 -15282.934} C_VEL
LIN {X 0,Y 327.669,Z 425.312,A -85,B 0,C 180,E1 -15284.448,E2 -15284.448} C_VEL
LIN {X 0,Y 325.957,Z 430.669,A -85,B 0,C 180,E1 -15286.28,E2 -15286.28} C_VEL
LIN {X 0,Y 323.975,Z 436.036,A -85,B 0,C 180,E1 -15288.741,E2 -15288.741} C_VEL
LIN {X 0,Y 323.164,Z 438.069,A -85,B 0,C 180,E1 -15289.98,E2 -15289.98} C_VEL
LIN {X 0,Y 322.457,Z 439.625,A -85,B 0,C 180,E1 -15291.224,E2 -15291.224} C_VEL
LIN {X 0,Y 321.765,Z 440.798,A -85,B 0,C 180,E1 -15292.469,E2 -15292.469} C_VEL
LIN {X 0,Y 321.23,Z 441.565,A -85,B 0,C 180,E1 -15293.72,E2 -15293.72} C_VEL
LIN {X 0,Y 320.783,Z 441.906,A -85,B 0,C 180,E1 -15294.972,E2 -15294.972} C_VEL
LIN {X 0,Y 320.127,Z 441.419,A -85,B 0,C 180,E1 -15297.483,E2 -15297.483} C_VEL
LIN {X 0,Y 319.933,Z 440.584,A -85,B 0,C 180,E1 -15298.741,E2 -15298.741} C_VEL
LIN {X 0,Y 319.838,Z 439.304,A -85,B 0,C 180,E1 -15300,E2 -15300} C_VEL
LIN {X 0,Y 319.683,Z 436.649,A -85,B 0,C 180,E1 -15301.89,E2 -15301.89} C_VEL
LIN {X 0,Y 319.5,Z 433.027,A -85,B 0,C 180,E1 -15303.784,E2 -15303.784} C_VEL
LIN {X 0,Y 320.029,Z 428.29,A -85,B 0,C 180,E1 -15305.671,E2 -15305.671} C_VEL
LIN {X 0,Y 320.447,Z 421.294,A -85,B 0,C 180,E1 -15307.878,E2 -15307.878} C_VEL
LIN {X 0,Y 321.04,Z 413.19,A -85,B 0,C 180,E1 -15309.897,E2 -15309.897} C_VEL
LIN {X 0,Y 321.677,Z 404.518,A -85,B 0,C 180,E1 -15311.659,E2 -15311.659} C_VEL
LIN {X 0,Y 322.522,Z 394.153,A -85,B 0,C 180,E1 -15313.387,E2 -15313.387} C_VEL
LIN {X 0,Y 323.365,Z 382.521,A -85,B 0,C 180,E1 -15314.957,E2 -15314.957} C_VEL
LIN {X 0,Y 323.874,Z 372.903,A -85,B 0,C 180,E1 -15316.031,E2 -15316.031} C_VEL
LIN {X 0,Y 320.89,Z 360.673,A -85,B 0,C 180,E1 -15317.279,E2 -15317.279} C_VEL
LIN {X 0,Y 319.671,Z 355.663,A -85,B 0,C 180,E1 -15317.719,E2 -15317.719} C_VEL
LIN {X 0,Y 319.614,Z 355.671,A -85,B 0,C 180,E1 -15320.599,E2 -15320.599} C_VEL
LIN {X 0,Y 319.573,Z 355.678,A -85,B 0,C 180,E1 -15323.319,E2 -15323.319} C_VEL
LIN {X 0,Y 319.637,Z 355.666,A -85,B 0,C 180,E1 -15326.088,E2 -15326.088} C_VEL
LIN {X 0,Y 319.592,Z 355.677,A -85,B 0,C 180,E1 -15328.933,E2 -15328.933} C_VEL
LIN {X 0,Y 319.534,Z 355.679,A -85,B 0,C 180,E1 -15331.861,E2 -15331.861} C_VEL
LIN {X 0,Y 319.582,Z 355.674,A -85,B 0,C 180,E1 -15335.543,E2 -15335.543} C_VEL
LIN {X 0,Y 319.584,Z 355.673,A -85,B 0,C 180,E1 -15338.006,E2 -15338.006} C_VEL
LIN {X 0,Y 319.573,Z 355.675,A -85,B 0,C 180,E1 -15341.606,E2 -15341.606} C_VEL
LIN {X 0,Y 319.522,Z 355.682,A -85,B 0,C 180,E1 -15345.263,E2 -15345.263} C_VEL
LIN {X 0,Y 319.53,Z 355.685,A -85,B 0,C 180,E1 -15348.712,E2 -15348.712} C_VEL
LIN {X 0,Y 319.579,Z 355.677,A -85,B 0,C 180,E1 -15352.344,E2 -15352.344} C_VEL
LIN {X 0,Y 319.561,Z 355.677,A -85,B 0,C 180,E1 -15355.123,E2 -15355.123} C_VEL
LIN {X 0,Y 319.567,Z 355.676,A -85,B 0,C 180,E1 -15359.059,E2 -15359.059} C_VEL
LIN {X 0,Y 319.607,Z 355.676,A -85,B 0,C 180,E1 -15362.498,E2 -15362.498} C_VEL
LIN {X 0,Y 319.606,Z 355.67,A -85,B 0,C 180,E1 -15365.304,E2 -15365.304} C_VEL
LIN {X 0,Y 319.623,Z 355.668,A -85,B 0,C 180,E1 -15369.402,E2 -15369.402} C_VEL
LIN {X 0,Y 319.66,Z 355.667,A -85,B 0,C 180,E1 -15372.073,E2 -15372.073} C_VEL
LIN {X 0,Y 319.733,Z 355.658,A -85,B 0,C 180,E1 -15376.008,E2 -15376.008} C_VEL
LIN {X 0,Y 319.753,Z 355.655,A -85,B 0,C 180,E1 -15379.873,E2 -15379.873} C_VEL
LIN {X 0,Y 319.913,Z 355.635,A -85,B 0,C 180,E1 -15382.426,E2 -15382.426} C_VEL
LIN {X 0,Y 319.746,Z 355.653,A -85,B 0,C 180,E1 -15384.956,E2 -15384.956} C_VEL
LIN {X 0,Y 319.992,Z 355.623,A -85,B 0,C 180,E1 -15387.482,E2 -15387.482} C_VEL
LIN {X 0,Y 320.15,Z 355.608,A -85,B 0,C 180,E1 -15390,E2 -15390} C_VEL
LIN {X 0,Y 319.993,Z 355.623,A -85,B 0,C 180,E1 -15392.518,E2 -15392.518} C_VEL
LIN {X 0,Y 319.944,Z 355.63,A -85,B 0,C 180,E1 -15396.306,E2 -15396.306} C_VEL
LIN {X 0,Y 319.838,Z 355.642,A -85,B 0,C 180,E1 -15398.848,E2 -15398.848} C_VEL
LIN {X 0,Y 319.682,Z 355.661,A -85,B 0,C 180,E1 -15402.7,E2 -15402.7} C_VEL
LIN {X 0,Y 319.7,Z 355.66,A -85,B 0,C 180,E1 -15405.296,E2 -15405.296} C_VEL
LIN {X 0,Y 319.676,Z 355.664,A -85,B 0,C 180,E1 -15409.255,E2 -15409.255} C_VEL
LIN {X 0,Y 319.572,Z 355.678,A -85,B 0,C 180,E1 -15413.32,E2 -15413.32} C_VEL
LIN {X 0,Y 319.635,Z 355.668,A -85,B 0,C 180,E1 -15416.088,E2 -15416.088} C_VEL
LIN {X 0,Y 319.581,Z 355.674,A -85,B 0,C 180,E1 -15418.935,E2 -15418.935} C_VEL
LIN {X 0,Y 319.531,Z 355.682,A -85,B 0,C 180,E1 -15421.862,E2 -15421.862} C_VEL
LIN {X 0,Y 319.581,Z 355.678,A -85,B 0,C 180,E1 -15425.543,E2 -15425.543} C_VEL
LIN {X 0,Y 319.583,Z 355.674,A -85,B 0,C 180,E1 -15428.007,E2 -15428.007} C_VEL
LIN {X 0,Y 319.598,Z 355.674,A -85,B 0,C 180,E1 -15431.612,E2 -15431.612} C_VEL
LIN {X 0,Y 319.566,Z 355.681,A -85,B 0,C 180,E1 -15435.271,E2 -15435.271} C_VEL
LIN {X 0,Y 319.53,Z 355.681,A -85,B 0,C 180,E1 -15438.712,E2 -15438.712} C_VEL
LIN {X 0,Y 319.556,Z 355.677,A -85,B 0,C 180,E1 -15442.35,E2 -15442.35} C_VEL
LIN {X 0,Y 319.563,Z 355.681,A -85,B 0,C 180,E1 -15445.124,E2 -15445.124} C_VEL
LIN {X 0,Y 319.573,Z 355.68,A -85,B 0,C 180,E1 -15449.058,E2 -15449.058} C_VEL
LIN {X 0,Y 319.612,Z 355.671,A -85,B 0,C 180,E1 -15452.499,E2 -15452.499} C_VEL
LIN {X 0,Y 319.608,Z 355.672,A -85,B 0,C 180,E1 -15455.304,E2 -15455.304} C_VEL
LIN {X 0,Y 319.601,Z 355.671,A -85,B 0,C 180,E1 -15458.048,E2 -15458.048} C_VEL
LIN {X 0,Y 319.692,Z 355.664,A -85,B 0,C 180,E1 -15460.963,E2 -15460.963} C_VEL
LIN {X 0,Y 319.735,Z 355.656,A -85,B 0,C 180,E1 -15465.276,E2 -15465.276} C_VEL
LIN {X 0,Y 319.698,Z 355.66,A -85,B 0,C 180,E1 -15468.207,E2 -15468.207} C_VEL
LIN {X 0,Y 319.129,Z 355.736,A -85,B 0,C 180,E1 -15469.259,E2 -15469.259} C_VEL
LIN {X 0,Y 316.467,Z 356.069,A -85,B 0,C 180,E1 -15470.977,E2 -15470.977} C_VEL
LIN {X 0,Y 313.272,Z 356.461,A -85,B 0,C 180,E1 -15473.08,E2 -15473.08} C_VEL
LIN {X 0,Y 312.864,Z 356.509,A -85,B 0,C 180,E1 -15473.805,E2 -15473.805} C_VEL
LIN {X 0,Y 312.94,Z 356.501,A -85,B 0,C 180,E1 -15477.426,E2 -15477.426} C_VEL
LIN {X 0,Y 313.106,Z 356.481,A -85,B 0,C 180,E1 -15480,E2 -15480} C_VEL
LIN {X 0,Y 312.942,Z 356.505,A -85,B 0,C 180,E1 -15482.575,E2 -15482.575} C_VEL
LIN {X 0,Y 312.897,Z 356.511,A -85,B 0,C 180,E1 -15486.448,E2 -15486.448} C_VEL
LIN {X 0,Y 312.702,Z 356.536,A -85,B 0,C 180,E1 -15490.358,E2 -15490.358} C_VEL
LIN {X 0,Y 312.704,Z 356.531,A -85,B 0,C 180,E1 -15494.888,E2 -15494.888} C_VEL
LIN {X 0,Y 312.635,Z 356.539,A -85,B 0,C 180,E1 -15499.237,E2 -15499.237} C_VEL
LIN {X 0,Y 312.55,Z 356.55,A -85,B 0,C 180,E1 -15502.789,E2 -15502.789} C_VEL
LIN {X 0,Y 312.607,Z 356.546,A -85,B 0,C 180,E1 -15505.936,E2 -15505.936} C_VEL
LIN {X 0,Y 312.549,Z 356.552,A -85,B 0,C 180,E1 -15509.65,E2 -15509.65} C_VEL
LIN {X 0,Y 312.523,Z 356.556,A -85,B 0,C 180,E1 -15513.689,E2 -15513.689} C_VEL
LIN {X 0,Y 312.541,Z 356.552,A -85,B 0,C 180,E1 -15517.383,E2 -15517.383} C_VEL
LIN {X 0,Y 312.496,Z 356.556,A -85,B 0,C 180,E1 -15520.709,E2 -15520.709} C_VEL
LIN {X 0,Y 312.53,Z 356.557,A -85,B 0,C 180,E1 -15522.753,E2 -15522.753} C_VEL
LIN {X 0,Y 314.206,Z 365.354,A -85,B 0,C 180,E1 -15526.705,E2 -15526.705} C_VEL
LIN {X 0,Y 315.991,Z 374.166,A -85,B 0,C 180,E1 -15530.486,E2 -15530.486} C_VEL
LIN {X 0,Y 316.593,Z 377.753,A -85,B 0,C 180,E1 -15531.974,E2 -15531.974} C_VEL
LIN {X 0,Y 315.763,Z 384.538,A -85,B 0,C 180,E1 -15534.641,E2 -15534.641} C_VEL
LIN {X 0,Y 314.238,Z 395.934,A -85,B 0,C 180,E1 -15539.042,E2 -15539.042} C_VEL
LIN {X 0,Y 313.053,Z 407.107,A -85,B 0,C 180,E1 -15543.32,E2 -15543.32} C_VEL
LIN {X 0,Y 312.156,Z 418.112,A -85,B 0,C 180,E1 -15547.496,E2 -15547.496} C_VEL
LIN {X 0,Y 311.856,Z 422.967,A -85,B 0,C 180,E1 -15549.339,E2 -15549.339} C_VEL
LIN {X 0,Y 312.577,Z 437.823,A -85,B 0,C 180,E1 -15550.119,E2 -15550.119} C_VEL
LIN {X 0,Y 313.263,Z 449.829,A -85,B 0,C 180,E1 -15550.978,E2 -15550.978} C_VEL
LIN {X 0,Y 313.968,Z 461.81,A -85,B 0,C 180,E1 -15552.074,E2 -15552.074} C_VEL
LIN {X 0,Y 314.444,Z 473.909,A -85,B 0,C 180,E1 -15553.443,E2 -15553.443} C_VEL
LIN {X 0,Y 313.422,Z 484.643,A -85,B 0,C 180,E1 -15554.949,E2 -15554.949} C_VEL
LIN {X 0,Y 312.641,Z 494.627,A -85,B 0,C 180,E1 -15556.678,E2 -15556.678} C_VEL
LIN {X 0,Y 312.124,Z 502.348,A -85,B 0,C 180,E1 -15558.308,E2 -15558.308} C_VEL
LIN {X 0,Y 311.853,Z 509.935,A -85,B 0,C 180,E1 -15560.269,E2 -15560.269} C_VEL
LIN {X 0,Y 311.944,Z 516.57,A -85,B 0,C 180,E1 -15562.442,E2 -15562.442} C_VEL
LIN {X 0,Y 312.161,Z 520.717,A -85,B 0,C 180,E1 -15564.185,E2 -15564.185} C_VEL
LIN {X 0,Y 312.349,Z 524.19,A -85,B 0,C 180,E1 -15566.129,E2 -15566.129} C_VEL
LIN {X 0,Y 312.5,Z 525.892,A -85,B 0,C 180,E1 -15567.422,E2 -15567.422} C_VEL
LIN {X 0,Y 312.65,Z 527.101,A -85,B 0,C 180,E1 -15568.712,E2 -15568.712} C_VEL
LIN {X 0,Y 312.836,Z 527.836,A -85,B 0,C 180,E1 -15570,E2 -15570} C_VEL
LIN {X 0,Y 312.555,Z 528.053,A -85,B 0,C 180,E1 -15571.288,E2 -15571.288} C_VEL
LIN {X 0,Y 312.159,Z 527.822,A -85,B 0,C 180,E1 -15572.581,E2 -15572.581} C_VEL
LIN {X 0,Y 311.994,Z 527.17,A -85,B 0,C 180,E1 -15573.875,E2 -15573.875} C_VEL
LIN {X 0,Y 311.794,Z 526.063,A -85,B 0,C 180,E1 -15575.173,E2 -15575.173} C_VEL
LIN {X 0,Y 311.479,Z 523.99,A -85,B 0,C 180,E1 -15576.884,E2 -15576.884} C_VEL
LIN {X 0,Y 311.351,Z 520.216,A -85,B 0,C 180,E1 -15579.091,E2 -15579.091} C_VEL
LIN {X 0,Y 311.566,Z 515.819,A -85,B 0,C 180,E1 -15581.054,E2 -15581.054} C_VEL
LIN {X 0,Y 312.372,Z 509.356,A -85,B 0,C 180,E1 -15583.333,E2 -15583.333} C_VEL
LIN {X 0,Y 313.695,Z 501.34,A -85,B 0,C 180,E1 -15585.596,E2 -15585.596} C_VEL
LIN {X 0,Y 315.462,Z 493.057,A -85,B 0,C 180,E1 -15587.503,E2 -15587.503} C_VEL
LIN {X 0,Y 317.735,Z 483.157,A -85,B 0,C 180,E1 -15589.377,E2 -15589.377} C_VEL
LIN {X 0,Y 319.531,Z 471.463,A -85,B 0,C 180,E1 -15591.279,E2 -15591.279} C_VEL
LIN {X 0,Y 321.112,Z 460.559,A -85,B 0,C 180,E1 -15592.78,E2 -15592.78} C_VEL
LIN {X 0,Y 321.733,Z 448.207,A -85,B 0,C 180,E1 -15594.35,E2 -15594.35} C_VEL
LIN {X 0,Y 321.087,Z 435.203,A -85,B 0,C 180,E1 -15595.961,E2 -15595.961} C_VEL
LIN {X 0,Y 319.291,Z 421.569,A -85,B 0,C 180,E1 -15597.67,E2 -15597.67} C_VEL
LIN {X 0,Y 316.781,Z 410.158,A -85,B 0,C 180,E1 -15599.215,E2 -15599.215} C_VEL
LIN {X 0,Y 315.74,Z 405.662,A -85,B 0,C 180,E1 -15599.84,E2 -15599.84} C_VEL
LIN {X 0,Y 314.434,Z 400.786,A -85,B 0,C 180,E1 -15600.563,E2 -15600.563} C_VEL
LIN {X 0,Y 314.357,Z 399.696,A -85,B 0,C 180,E1 -15600.711,E2 -15600.711} C_VEL
LIN {X 0,Y 315.862,Z 390.639,A -85,B 0,C 180,E1 -15604.587,E2 -15604.587} C_VEL
LIN {X 0,Y 317.701,Z 382.722,A -85,B 0,C 180,E1 -15608.273,E2 -15608.273} C_VEL
LIN {X 0,Y 317.377,Z 379.733,A -85,B 0,C 180,E1 -15609.955,E2 -15609.955} C_VEL
LIN {X 0,Y 316.582,Z 375.096,A -85,B 0,C 180,E1 -15612.896,E2 -15612.896} C_VEL
LIN {X 0,Y 315.574,Z 370.564,A -85,B 0,C 180,E1 -15616.339,E2 -15616.339} C_VEL
LIN {X 0,Y 314.818,Z 367.001,A -85,B 0,C 180,E1 -15619.654,E2 -15619.654} C_VEL
LIN {X 0,Y 314.096,Z 363.7,A -85,B 0,C 180,E1 -15623.66,E2 -15623.66} C_VEL
LIN {X 0,Y 313.616,Z 361.513,A -85,B 0,C 180,E1 -15627.464,E2 -15627.464} C_VEL
LIN {X 0,Y 313.556,Z 361.144,A -85,B 0,C 180,E1 -15628.401,E2 -15628.401} C_VEL
LIN {X 0,Y 314.968,Z 363.401,A -85,B 0,C 180,E1 -15629.122,E2 -15629.122} C_VEL
LIN {X 0,Y 316.889,Z 364.784,A -85,B 0,C 180,E1 -15629.877,E2 -15629.877} C_VEL
LIN {X 0,Y 321.042,Z 370.47,A -85,B 0,C 180,E1 -15631.713,E2 -15631.713} C_VEL
LIN {X 0,Y 324.898,Z 378.47,A -85,B 0,C 180,E1 -15633.7,E2 -15633.7} C_VEL
LIN {X 0,Y 328.124,Z 387.283,A -85,B 0,C 180,E1 -15635.692,E2 -15635.692} C_VEL
LIN {X 0,Y 329.795,Z 393.732,A -85,B 0,C 180,E1 -15637.092,E2 -15637.092} C_VEL
LIN {X 0,Y 329.987,Z 395.611,A -85,B 0,C 180,E1 -15637.458,E2 -15637.458} C_VEL
LIN {X 0,Y 327.675,Z 405.18,A -85,B 0,C 180,E1 -15638.945,E2 -15638.945} C_VEL
LIN {X 0,Y 325.185,Z 414.588,A -85,B 0,C 180,E1 -15640.756,E2 -15640.756} C_VEL
LIN {X 0,Y 322.881,Z 422.216,A -85,B 0,C 180,E1 -15642.585,E2 -15642.585} C_VEL
LIN {X 0,Y 320.485,Z 429.42,A -85,B 0,C 180,E1 -15644.773,E2 -15644.773} C_VEL
LIN {X 0,Y 318.839,Z 434.102,A -85,B 0,C 180,E1 -15646.618,E2 -15646.618} C_VEL
LIN {X 0,Y 317.249,Z 437.805,A -85,B 0,C 180,E1 -15648.499,E2 -15648.499} C_VEL
LIN {X 0,Y 315.604,Z 441.14,A -85,B 0,C 180,E1 -15651.032,E2 -15651.032} C_VEL
LIN {X 0,Y 314.875,Z 442.243,A -85,B 0,C 180,E1 -15652.304,E2 -15652.304} C_VEL
LIN {X 0,Y 314.299,Z 442.905,A -85,B 0,C 180,E1 -15653.58,E2 -15653.58} C_VEL
LIN {X 0,Y 313.423,Z 443.029,A -85,B 0,C 180,E1 -15656.143,E2 -15656.143} C_VEL
LIN {X 0,Y 313.117,Z 442.51,A -85,B 0,C 180,E1 -15657.427,E2 -15657.427} C_VEL
LIN {X 0,Y 312.912,Z 441.555,A -85,B 0,C 180,E1 -15658.713,E2 -15658.713} C_VEL
LIN {X 0,Y 312.813,Z 440.198,A -85,B 0,C 180,E1 -15660,E2 -15660} C_VEL
LIN {X 0,Y 312.639,Z 437.411,A -85,B 0,C 180,E1 -15661.932,E2 -15661.932} C_VEL
LIN {X 0,Y 312.459,Z 433.646,A -85,B 0,C 180,E1 -15663.869,E2 -15663.869} C_VEL
LIN {X 0,Y 312.99,Z 428.757,A -85,B 0,C 180,E1 -15665.799,E2 -15665.799} C_VEL
LIN {X 0,Y 313.419,Z 421.577,A -85,B 0,C 180,E1 -15668.056,E2 -15668.056} C_VEL
LIN {X 0,Y 314.014,Z 413.771,A -85,B 0,C 180,E1 -15670.01,E2 -15670.01} C_VEL
LIN {X 0,Y 314.704,Z 404.464,A -85,B 0,C 180,E1 -15671.921,E2 -15671.921} C_VEL
LIN {X 0,Y 315.597,Z 393.807,A -85,B 0,C 180,E1 -15673.686,E2 -15673.686} C_VEL
LIN {X 0,Y 316.462,Z 381.891,A -85,B 0,C 180,E1 -15675.291,E2 -15675.291} C_VEL
LIN {X 0,Y 316.914,Z 374.297,A -85,B 0,C 180,E1 -15676.142,E2 -15676.142} C_VEL
LIN {X 0,Y 313.981,Z 362.19,A -85,B 0,C 180,E1 -15677.42,E2 -15677.42} C_VEL
LIN {X 0,Y 312.626,Z 356.538,A -85,B 0,C 180,E1 -15677.963,E2 -15677.963} C_VEL
LIN {X 0,Y 312.59,Z 356.545,A -85,B 0,C 180,E1 -15682.471,E2 -15682.471} C_VEL
LIN {X 0,Y 312.605,Z 356.542,A -85,B 0,C 180,E1 -15685.935,E2 -15685.935} C_VEL
LIN {X 0,Y 312.547,Z 356.55,A -85,B 0,C 180,E1 -15689.65,E2 -15689.65} C_VEL
LIN {X 0,Y 312.521,Z 356.553,A -85,B 0,C 180,E1 -15693.689,E2 -15693.689} C_VEL
LIN {X 0,Y 312.542,Z 356.552,A -85,B 0,C 180,E1 -15697.383,E2 -15697.383} C_VEL
LIN {X 0,Y 312.503,Z 356.56,A -85,B 0,C 180,E1 -15700.707,E2 -15700.707} C_VEL
LIN {X 0,Y 312.518,Z 356.554,A -85,B 0,C 180,E1 -15704.198,E2 -15704.198} C_VEL
LIN {X 0,Y 312.487,Z 356.558,A -85,B 0,C 180,E1 -15707.918,E2 -15707.918} C_VEL
LIN {X 0,Y 312.536,Z 356.551,A -85,B 0,C 180,E1 -15711.91,E2 -15711.91} C_VEL
LIN {X 0,Y 312.507,Z 356.555,A -85,B 0,C 180,E1 -15715.79,E2 -15715.79} C_VEL
LIN {X 0,Y 312.521,Z 356.555,A -85,B 0,C 180,E1 -15718.853,E2 -15718.853} C_VEL
LIN {X 0,Y 312.571,Z 356.547,A -85,B 0,C 180,E1 -15721.824,E2 -15721.824} C_VEL
LIN {X 0,Y 312.586,Z 356.548,A -85,B 0,C 180,E1 -15724.711,E2 -15724.711} C_VEL
LIN {X 0,Y 312.588,Z 356.545,A -85,B 0,C 180,E1 -15727.529,E2 -15727.529} C_VEL
LIN {X 0,Y 312.64,Z 356.539,A -85,B 0,C 180,E1 -15731.656,E2 -15731.656} C_VEL
LIN {X 0,Y 312.694,Z 356.532,A -85,B 0,C 180,E1 -15735.686,E2 -15735.686} C_VEL
LIN {X 0,Y 312.699,Z 356.532,A -85,B 0,C 180,E1 -15739.642,E2 -15739.642} C_VEL
LIN {X 0,Y 312.854,Z 356.516,A -85,B 0,C 180,E1 -15742.254,E2 -15742.254} C_VEL
LIN {X 0,Y 312.716,Z 356.529,A -85,B 0,C 180,E1 -15744.842,E2 -15744.842} C_VEL
LIN {X 0,Y 312.99,Z 356.495,A -85,B 0,C 180,E1 -15748.713,E2 -15748.713} C_VEL
LIN {X 0,Y 312.992,Z 356.495,A -85,B 0,C 180,E1 -15751.287,E2 -15751.287} C_VEL
LIN {X 0,Y 312.717,Z 356.529,A -85,B 0,C 180,E1 -15755.158,E2 -15755.158} C_VEL
LIN {X 0,Y 312.854,Z 356.516,A -85,B 0,C 180,E1 -15757.746,E2 -15757.746} C_VEL
LIN {X 0,Y 312.67,Z 356.539,A -85,B 0,C 180,E1 -15761.671,E2 -15761.671} C_VEL
LIN {X 0,Y 312.701,Z 356.531,A -85,B 0,C 180,E1 -15764.888,E2 -15764.888} C_VEL
LIN {X 0,Y 312.632,Z 356.541,A -85,B 0,C 180,E1 -15769.237,E2 -15769.237} C_VEL
LIN {X 0,Y 312.547,Z 356.55,A -85,B 0,C 180,E1 -15772.79,E2 -15772.79} C_VEL
LIN {X 0,Y 312.603,Z 356.545,A -85,B 0,C 180,E1 -15775.936,E2 -15775.936} C_VEL
LIN {X 0,Y 312.539,Z 356.555,A -85,B 0,C 180,E1 -15779.651,E2 -15779.651} C_VEL
LIN {X 0,Y 312.52,Z 356.556,A -85,B 0,C 180,E1 -15783.689,E2 -15783.689} C_VEL
LIN {X 0,Y 312.541,Z 356.556,A -85,B 0,C 180,E1 -15787.383,E2 -15787.383} C_VEL
LIN {X 0,Y 312.528,Z 356.553,A -85,B 0,C 180,E1 -15790.704,E2 -15790.704} C_VEL
LIN {X 0,Y 312.532,Z 356.552,A -85,B 0,C 180,E1 -15794.196,E2 -15794.196} C_VEL
LIN {X 0,Y 312.489,Z 356.557,A -85,B 0,C 180,E1 -15797.918,E2 -15797.918} C_VEL
LIN {X 0,Y 312.5,Z 356.559,A -85,B 0,C 180,E1 -15800.972,E2 -15800.972} C_VEL
LIN {X 0,Y 312.534,Z 356.551,A -85,B 0,C 180,E1 -15804.221,E2 -15804.221} C_VEL
LIN {X 0,Y 312.507,Z 356.558,A -85,B 0,C 180,E1 -15807.334,E2 -15807.334} C_VEL
LIN {X 0,Y 312.555,Z 356.551,A -85,B 0,C 180,E1 -15811.276,E2 -15811.276} C_VEL
LIN {X 0,Y 312.589,Z 356.548,A -85,B 0,C 180,E1 -15814.711,E2 -15814.711} C_VEL
LIN {X 0,Y 312.591,Z 356.545,A -85,B 0,C 180,E1 -15817.529,E2 -15817.529} C_VEL
LIN {X 0,Y 312.642,Z 356.538,A -85,B 0,C 180,E1 -15821.657,E2 -15821.657} C_VEL
LIN {X 0,Y 312.698,Z 356.531,A -85,B 0,C 180,E1 -15825.687,E2 -15825.687} C_VEL
LIN {X 0,Y 312.706,Z 356.53,A -85,B 0,C 180,E1 -15829.642,E2 -15829.642} C_VEL
LIN {X 0,Y 312.876,Z 356.511,A -85,B 0,C 180,E1 -15832.255,E2 -15832.255} C_VEL
LIN {X 0,Y 312.864,Z 356.509,A -85,B 0,C 180,E1 -15833.805,E2 -15833.805} C_VEL
LIN {X 0,Y 312.074,Z 356.612,A -85,B 0,C 180,E1 -15834.88,E2 -15834.88} C_VEL
LIN {X 0,Y 309.24,Z 356.966,A -85,B 0,C 180,E1 -15836.632,E2 -15836.632} C_VEL
LIN {X 0,Y 306.962,Z 357.248,A -85,B 0,C 180,E1 -15838.053,E2 -15838.053} C_VEL
LIN {X 0,Y 306.049,Z 357.36,A -85,B 0,C 180,E1 -15839.151,E2 -15839.151} C_VEL
LIN {X 0,Y 306.004,Z 357.364,A -85,B 0,C 180,E1 -15839.522,E2 -15839.522} C_VEL
LIN {X 0,Y 305.891,Z 357.383,A -85,B 0,C 180,E1 -15842.634,E2 -15842.634} C_VEL
LIN {X 0,Y 305.837,Z 357.389,A -85,B 0,C 180,E1 -15846.598,E2 -15846.598} C_VEL
LIN {X 0,Y 305.702,Z 357.402,A -85,B 0,C 180,E1 -15849.261,E2 -15849.261} C_VEL
LIN {X 0,Y 305.593,Z 357.416,A -85,B 0,C 180,E1 -15853.296,E2 -15853.296} C_VEL
LIN {X 0,Y 305.598,Z 357.419,A -85,B 0,C 180,E1 -15856.02,E2 -15856.02} C_VEL
LIN {X 0,Y 305.581,Z 357.418,A -85,B 0,C 180,E1 -15859.445,E2 -15859.445} C_VEL
LIN {X 0,Y 305.495,Z 357.428,A -85,B 0,C 180,E1 -15863.041,E2 -15863.041} C_VEL
LIN {X 0,Y 305.552,Z 357.425,A -85,B 0,C 180,E1 -15866.227,E2 -15866.227} C_VEL
LIN {X 0,Y 305.499,Z 357.428,A -85,B 0,C 180,E1 -15869.05,E2 -15869.05} C_VEL
LIN {X 0,Y 305.449,Z 357.439,A -85,B 0,C 180,E1 -15871.952,E2 -15871.952} C_VEL
LIN {X 0,Y 305.466,Z 357.432,A -85,B 0,C 180,E1 -15875.113,E2 -15875.113} C_VEL
LIN {X 0,Y 305.47,Z 357.432,A -85,B 0,C 180,E1 -15878.533,E2 -15878.533} C_VEL
LIN {X 0,Y 305.51,Z 357.616,A -85,B 0,C 180,E1 -15882.596,E2 -15882.596} C_VEL
LIN {X 0,Y 307.213,Z 366.464,A -85,B 0,C 180,E1 -15886.662,E2 -15886.662} C_VEL
LIN {X 0,Y 309.037,Z 375.53,A -85,B 0,C 180,E1 -15890.644,E2 -15890.644} C_VEL
LIN {X 0,Y 309.531,Z 379.216,A -85,B 0,C 180,E1 -15892.19,E2 -15892.19} C_VEL
LIN {X 0,Y 308.444,Z 386.906,A -85,B 0,C 180,E1 -15895.275,E2 -15895.275} C_VEL
LIN {X 0,Y 307.154,Z 396.341,A -85,B 0,C 180,E1 -15899.014,E2 -15899.014} C_VEL
LIN {X 0,Y 305.975,Z 407.047,A -85,B 0,C 180,E1 -15903.219,E2 -15903.219} C_VEL
LIN {X 0,Y 305.125,Z 417.027,A -85,B 0,C 180,E1 -15907.122,E2 -15907.122} C_VEL
LIN {X 0,Y 304.802,Z 422.24,A -85,B 0,C 180,E1 -15909.104,E2 -15909.104} C_VEL
LIN {X 0,Y 305.394,Z 435.466,A -85,B 0,C 180,E1 -15909.806,E2 -15909.806} C_VEL
LIN {X 0,Y 306.117,Z 449.07,A -85,B 0,C 180,E1 -15910.794,E2 -15910.794} C_VEL
LIN {X 0,Y 306.856,Z 461.677,A -85,B 0,C 180,E1 -15911.989,E2 -15911.989} C_VEL
LIN {X 0,Y 307.343,Z 473.613,A -85,B 0,C 180,E1 -15913.391,E2 -15913.391} C_VEL
LIN {X 0,Y 306.37,Z 483.828,A -85,B 0,C 180,E1 -15914.878,E2 -15914.878} C_VEL
LIN {X 0,Y 305.582,Z 494.039,A -85,B 0,C 180,E1 -15916.703,E2 -15916.703} C_VEL
LIN {X 0,Y 305.037,Z 503.019,A -85,B 0,C 180,E1 -15918.706,E2 -15918.706} C_VEL
LIN {X 0,Y 304.827,Z 510.245,A -85,B 0,C 180,E1 -15920.712,E2 -15920.712} C_VEL
LIN {X 0,Y 304.984,Z 516.106,A -85,B 0,C 180,E1 -15922.748,E2 -15922.748} C_VEL
LIN {X 0,Y 305.216,Z 520.474,A -85,B 0,C 180,E1 -15924.715,E2 -15924.715} C_VEL
LIN {X 0,Y 305.353,Z 522.723,A -85,B 0,C 180,E1 -15926.041,E2 -15926.041} C_VEL
LIN {X 0,Y 305.517,Z 524.482,A -85,B 0,C 180,E1 -15927.363,E2 -15927.363} C_VEL
LIN {X 0,Y 305.651,Z 525.774,A -85,B 0,C 180,E1 -15928.682,E2 -15928.682} C_VEL
LIN {X 0,Y 305.862,Z 526.593,A -85,B 0,C 180,E1 -15930,E2 -15930} C_VEL
LIN {X 0,Y 305.536,Z 526.854,A -85,B 0,C 180,E1 -15931.318,E2 -15931.318} C_VEL
LIN {X 0,Y 304.941,Z 526.103,A -85,B 0,C 180,E1 -15933.965,E2 -15933.965} C_VEL
LIN {X 0,Y 304.715,Z 525.082,A -85,B 0,C 180,E1 -15935.293,E2 -15935.293} C_VEL
LIN {X 0,Y 304.321,Z 521.728,A -85,B 0,C 180,E1 -15937.965,E2 -15937.965} C_VEL
LIN {X 0,Y 304.415,Z 516.731,A -85,B 0,C 180,E1 -15940.643,E2 -15940.643} C_VEL
LIN {X 0,Y 305.26,Z 509.92,A -85,B 0,C 180,E1 -15943.311,E2 -15943.311} C_VEL
LIN {X 0,Y 306.617,Z 502.141,A -85,B 0,C 180,E1 -15945.7,E2 -15945.7} C_VEL
LIN {X 0,Y 308.693,Z 493.148,A -85,B 0,C 180,E1 -15947.9,E2 -15947.9} C_VEL
LIN {X 0,Y 311.065,Z 483.636,A -85,B 0,C 180,E1 -15949.81,E2 -15949.81} C_VEL
LIN {X 0,Y 313.002,Z 472.411,A -85,B 0,C 180,E1 -15951.746,E2 -15951.746} C_VEL
LIN {X 0,Y 314.875,Z 460.832,A -85,B 0,C 180,E1 -15953.433,E2 -15953.433} C_VEL
LIN {X 0,Y 315.609,Z 449.11,A -85,B 0,C 180,E1 -15955.03,E2 -15955.03} C_VEL
LIN {X 0,Y 315.239,Z 437.033,A -85,B 0,C 180,E1 -15956.639,E2 -15956.639} C_VEL
LIN {X 0,Y 313.967,Z 424.878,A -85,B 0,C 180,E1 -15958.275,E2 -15958.275} C_VEL
LIN {X 0,Y 311.224,Z 410.121,A -85,B 0,C 180,E1 -15960.419,E2 -15960.419} C_VEL
LIN {X 0,Y 309.172,Z 402.267,A -85,B 0,C 180,E1 -15961.715,E2 -15961.715} C_VEL
LIN {X 0,Y 308.099,Z 397.57,A -85,B 0,C 180,E1 -15962.486,E2 -15962.486} C_VEL
LIN {X 0,Y 308.081,Z 396.615,A -85,B 0,C 180,E1 -15962.702,E2 -15962.702} C_VEL
LIN {X 0,Y 310.014,Z 387.5,A -85,B 0,C 180,E1 -15966.884,E2 -15966.884} C_VEL
LIN {X 0,Y 310.838,Z 384.333,A -85,B 0,C 180,E1 -15968.446,E2 -15968.446} C_VEL
LIN {X 0,Y 310.275,Z 379.933,A -85,B 0,C 180,E1 -15971.062,E2 -15971.062} C_VEL
LIN {X 0,Y 309.662,Z 376.44,A -85,B 0,C 180,E1 -15973.426,E2 -15973.426} C_VEL
LIN {X 0,Y 308.692,Z 372.058,A -85,B 0,C 180,E1 -15976.92,E2 -15976.92} C_VEL
LIN {X 0,Y 307.807,Z 368.079,A -85,B 0,C 180,E1 -15980.924,E2 -15980.924} C_VEL
LIN {X 0,Y 307.378,Z 366.045,A -85,B 0,C 180,E1 -15983.525,E2 -15983.525} C_VEL
LIN {X 0,Y 307.015,Z 364.342,A -85,B 0,C 180,E1 -15986.373,E2 -15986.373} C_VEL
LIN {X 0,Y 307.491,Z 365.369,A -85,B 0,C 180,E1 -15986.733,E2 -15986.733} C_VEL
LIN {X 0,Y 308.693,Z 366.653,A -85,B 0,C 180,E1 -15987.393,E2 -15987.393} C_VEL
LIN {X 0,Y 310.341,Z 367.539,A -85,B 0,C 180,E1 -15988.139,E2 -15988.139} C_VEL
LIN {X 0,Y 311.778,Z 369.653,A -85,B 0,C 180,E1 -15988.936,E2 -15988.936} C_VEL
LIN {X 0,Y 313.353,Z 370.825,A -85,B 0,C 180,E1 -15989.62,E2 -15989.62} C_VEL
LIN {X 0,Y 316.916,Z 376.019,A -85,B 0,C 180,E1 -15991.406,E2 -15991.406} C_VEL
LIN {X 0,Y 320.587,Z 384.5,A -85,B 0,C 180,E1 -15993.639,E2 -15993.639} C_VEL
LIN {X 0,Y 323.439,Z 393.87,A -85,B 0,C 180,E1 -15995.87,E2 -15995.87} C_VEL
LIN {X 0,Y 324.195,Z 397.681,A -85,B 0,C 180,E1 -15996.745,E2 -15996.745} C_VEL
LIN {X 0,Y 322.538,Z 404.919,A -85,B 0,C 180,E1 -15997.922,E2 -15997.922} C_VEL
LIN {X 0,Y 319.796,Z 414.538,A -85,B 0,C 180,E1 -15999.749,E2 -15999.749} C_VEL
LIN {X 0,Y 317.291,Z 422.387,A -85,B 0,C 180,E1 -16001.6,E2 -16001.6} C_VEL
LIN {X 0,Y 314.984,Z 428.883,A -85,B 0,C 180,E1 -16003.513,E2 -16003.513} C_VEL
LIN {X 0,Y 312.751,Z 434.611,A -85,B 0,C 180,E1 -16005.689,E2 -16005.689} C_VEL
LIN {X 0,Y 311.089,Z 438.458,A -85,B 0,C 180,E1 -16007.607,E2 -16007.607} C_VEL
LIN {X 0,Y 309.581,Z 441.331,A -85,B 0,C 180,E1 -16009.536,E2 -16009.536} C_VEL
LIN {X 0,Y 308.788,Z 442.704,A -85,B 0,C 180,E1 -16010.832,E2 -16010.832} C_VEL
LIN {X 0,Y 307.987,Z 443.681,A -85,B 0,C 180,E1 -16012.13,E2 -16012.13} C_VEL
LIN {X 0,Y 306.856,Z 444.399,A -85,B 0,C 180,E1 -16014.743,E2 -16014.743} C_VEL
LIN {X 0,Y 306.434,Z 444.195,A -85,B 0,C 180,E1 -16016.054,E2 -16016.054} C_VEL
LIN {X 0,Y 306.103,Z 443.557,A -85,B 0,C 180,E1 -16017.368,E2 -16017.368} C_VEL
LIN {X 0,Y 305.787,Z 441.078,A -85,B 0,C 180,E1 -16020,E2 -16020} C_VEL
LIN {X 0,Y 305.594,Z 438.153,A -85,B 0,C 180,E1 -16021.977,E2 -16021.977} C_VEL
LIN {X 0,Y 305.42,Z 434.249,A -85,B 0,C 180,E1 -16023.958,E2 -16023.958} C_VEL
LIN {X 0,Y 305.956,Z 429.205,A -85,B 0,C 180,E1 -16025.933,E2 -16025.933} C_VEL
LIN {X 0,Y 306.39,Z 421.791,A -85,B 0,C 180,E1 -16028.242,E2 -16028.242} C_VEL
LIN {X 0,Y 306.971,Z 414.363,A -85,B 0,C 180,E1 -16030.109,E2 -16030.109} C_VEL
LIN {X 0,Y 307.591,Z 405.958,A -85,B 0,C 180,E1 -16031.867,E2 -16031.867} C_VEL
LIN {X 0,Y 308.453,Z 395.443,A -85,B 0,C 180,E1 -16033.673,E2 -16033.673} C_VEL
LIN {X 0,Y 309.351,Z 383.724,A -85,B 0,C 180,E1 -16035.313,E2 -16035.313} C_VEL
LIN {X 0,Y 309.911,Z 375.766,A -85,B 0,C 180,E1 -16036.239,E2 -16036.239} C_VEL
LIN {X 0,Y 307.031,Z 363.437,A -85,B 0,C 180,E1 -16037.569,E2 -16037.569} C_VEL
LIN {X 0,Y 305.605,Z 357.411,A -85,B 0,C 180,E1 -16038.13,E2 -16038.13} C_VEL
LIN {X 0,Y 305.502,Z 357.429,A -85,B 0,C 180,E1 -16041.597,E2 -16041.597} C_VEL
LIN {X 0,Y 305.574,Z 357.418,A -85,B 0,C 180,E1 -16045.912,E2 -16045.912} C_VEL
LIN {X 0,Y 305.498,Z 357.433,A -85,B 0,C 180,E1 -16049.05,E2 -16049.05} C_VEL
LIN {X 0,Y 305.467,Z 357.432,A -85,B 0,C 180,E1 -16053.516,E2 -16053.516} C_VEL
LIN {X 0,Y 305.499,Z 357.432,A -85,B 0,C 180,E1 -16056.736,E2 -16056.736} C_VEL
LIN {X 0,Y 305.465,Z 357.435,A -85,B 0,C 180,E1 -16060.602,E2 -16060.602} C_VEL
LIN {X 0,Y 305.481,Z 357.43,A -85,B 0,C 180,E1 -16063.645,E2 -16063.645} C_VEL
LIN {X 0,Y 305.46,Z 357.433,A -85,B 0,C 180,E1 -16067.413,E2 -16067.413} C_VEL
LIN {X 0,Y 305.496,Z 357.428,A -85,B 0,C 180,E1 -16071.6,E2 -16071.6} C_VEL
LIN {X 0,Y 305.463,Z 357.435,A -85,B 0,C 180,E1 -16074.887,E2 -16074.887} C_VEL
LIN {X 0,Y 305.45,Z 357.438,A -85,B 0,C 180,E1 -16078.355,E2 -16078.355} C_VEL
LIN {X 0,Y 305.513,Z 357.426,A -85,B 0,C 180,E1 -16081.113,E2 -16081.113} C_VEL
LIN {X 0,Y 305.571,Z 357.421,A -85,B 0,C 180,E1 -16084.088,E2 -16084.088} C_VEL
LIN {X 0,Y 305.53,Z 357.429,A -85,B 0,C 180,E1 -16088.405,E2 -16088.405} C_VEL
LIN {X 0,Y 305.592,Z 357.416,A -85,B 0,C 180,E1 -16091.218,E2 -16091.218} C_VEL
LIN {X 0,Y 305.649,Z 357.409,A -85,B 0,C 180,E1 -16095.349,E2 -16095.349} C_VEL
LIN {X 0,Y 305.636,Z 357.411,A -85,B 0,C 180,E1 -16099.4,E2 -16099.4} C_VEL
LIN {X 0,Y 305.798,Z 357.396,A -85,B 0,C 180,E1 -16102.074,E2 -16102.074} C_VEL
LIN {X 0,Y 305.687,Z 357.405,A -85,B 0,C 180,E1 -16104.723,E2 -16104.723} C_VEL
LIN {X 0,Y 305.957,Z 357.371,A -85,B 0,C 180,E1 -16108.684,E2 -16108.684} C_VEL
LIN {X 0,Y 305.958,Z 357.371,A -85,B 0,C 180,E1 -16111.316,E2 -16111.316} C_VEL
LIN {X 0,Y 305.688,Z 357.404,A -85,B 0,C 180,E1 -16115.277,E2 -16115.277} C_VEL
LIN {X 0,Y 305.798,Z 357.396,A -85,B 0,C 180,E1 -16117.926,E2 -16117.926} C_VEL
LIN {X 0,Y 305.604,Z 357.418,A -85,B 0,C 180,E1 -16121.945,E2 -16121.945} C_VEL
LIN {X 0,Y 305.638,Z 357.411,A -85,B 0,C 180,E1 -16125.035,E2 -16125.035} C_VEL
LIN {X 0,Y 305.578,Z 357.421,A -85,B 0,C 180,E1 -16129.445,E2 -16129.445} C_VEL
LIN {X 0,Y 305.492,Z 357.429,A -85,B 0,C 180,E1 -16133.042,E2 -16133.042} C_VEL
LIN {X 0,Y 305.532,Z 357.424,A -85,B 0,C 180,E1 -16136.221,E2 -16136.221} C_VEL
LIN {X 0,Y 305.489,Z 357.43,A -85,B 0,C 180,E1 -16139.048,E2 -16139.048} C_VEL
LIN {X 0,Y 305.443,Z 357.436,A -85,B 0,C 180,E1 -16141.953,E2 -16141.953} C_VEL
LIN {X 0,Y 305.464,Z 357.435,A -85,B 0,C 180,E1 -16145.113,E2 -16145.113} C_VEL
LIN {X 0,Y 305.484,Z 357.429,A -85,B 0,C 180,E1 -16148.537,E2 -16148.537} C_VEL
LIN {X 0,Y 305.51,Z 357.427,A -85,B 0,C 180,E1 -16152.597,E2 -16152.597} C_VEL
LIN {X 0,Y 305.472,Z 357.431,A -85,B 0,C 180,E1 -16156.353,E2 -16156.353} C_VEL
LIN {X 0,Y 305.46,Z 357.433,A -85,B 0,C 180,E1 -16159.893,E2 -16159.893} C_VEL
LIN {X 0,Y 305.482,Z 357.431,A -85,B 0,C 180,E1 -16163.632,E2 -16163.632} C_VEL
LIN {X 0,Y 305.467,Z 357.432,A -85,B 0,C 180,E1 -16166.484,E2 -16166.484} C_VEL
LIN {X 0,Y 305.499,Z 357.433,A -85,B 0,C 180,E1 -16170.95,E2 -16170.95} C_VEL
LIN {X 0,Y 305.575,Z 357.418,A -85,B 0,C 180,E1 -16174.088,E2 -16174.088} C_VEL
LIN {X 0,Y 305.504,Z 357.429,A -85,B 0,C 180,E1 -16178.403,E2 -16178.403} C_VEL
LIN {X 0,Y 305.594,Z 357.418,A -85,B 0,C 180,E1 -16181.218,E2 -16181.218} C_VEL
LIN {X 0,Y 305.653,Z 357.409,A -85,B 0,C 180,E1 -16185.349,E2 -16185.349} C_VEL
LIN {X 0,Y 305.643,Z 357.41,A -85,B 0,C 180,E1 -16189.4,E2 -16189.4} C_VEL
LIN {X 0,Y 305.817,Z 357.389,A -85,B 0,C 180,E1 -16192.075,E2 -16192.075} C_VEL
LIN {X 0,Y 305.692,Z 357.408,A -85,B 0,C 180,E1 -16194.724,E2 -16194.724} C_VEL
LIN {X 0,Y 305.96,Z 357.374,A -85,B 0,C 180,E1 -16198.684,E2 -16198.684} C_VEL
LIN {X 0,Y 306.004,Z 357.364,A -85,B 0,C 180,E1 -16199.522,E2 -16199.522} C_VEL
LIN {X 0,Y 305.361,Z 357.449,A -85,B 0,C 180,E1 -16200.62,E2 -16200.62} C_VEL
LIN {X 0,Y 302.333,Z 357.827,A -85,B 0,C 180,E1 -16202.399,E2 -16202.399} C_VEL
LIN {X 0,Y 299.761,Z 358.144,A -85,B 0,C 180,E1 -16203.845,E2 -16203.845} C_VEL
LIN {X 0,Y 298.708,Z 358.275,A -85,B 0,C 180,E1 -16204.969,E2 -16204.969} C_VEL
LIN {X 0,Y 298.653,Z 358.28,A -85,B 0,C 180,E1 -16205.35,E2 -16205.35} C_VEL
LIN {X 0,Y 298.722,Z 358.275,A -85,B 0,C 180,E1 -16208.115,E2 -16208.115} C_VEL
LIN {X 0,Y 298.558,Z 358.297,A -85,B 0,C 180,E1 -16212.232,E2 -16212.232} C_VEL
LIN {X 0,Y 298.61,Z 358.286,A -85,B 0,C 180,E1 -16215.209,E2 -16215.209} C_VEL
LIN {X 0,Y 298.544,Z 358.294,A -85,B 0,C 180,E1 -16219.243,E2 -16219.243} C_VEL
LIN {X 0,Y 298.461,Z 358.306,A -85,B 0,C 180,E1 -16223.598,E2 -16223.598} C_VEL
LIN {X 0,Y 298.493,Z 358.301,A -85,B 0,C 180,E1 -16226.574,E2 -16226.574} C_VEL
LIN {X 0,Y 298.425,Z 358.311,A -85,B 0,C 180,E1 -16229.641,E2 -16229.641} C_VEL
LIN {X 0,Y 298.4,Z 358.312,A -85,B 0,C 180,E1 -16232.8,E2 -16232.8} C_VEL
LIN {X 0,Y 298.468,Z 358.304,A -85,B 0,C 180,E1 -16236.812,E2 -16236.812} C_VEL
LIN {X 0,Y 298.418,Z 358.311,A -85,B 0,C 180,E1 -16241.256,E2 -16241.256} C_VEL
LIN {X 0,Y 298.476,Z 358.52,A -85,B 0,C 180,E1 -16242.378,E2 -16242.378} C_VEL
LIN {X 0,Y 300.156,Z 367.355,A -85,B 0,C 180,E1 -16246.54,E2 -16246.54} C_VEL
LIN {X 0,Y 302.037,Z 376.566,A -85,B 0,C 180,E1 -16250.667,E2 -16250.667} C_VEL
LIN {X 0,Y 302.46,Z 380.091,A -85,B 0,C 180,E1 -16252.189,E2 -16252.189} C_VEL
LIN {X 0,Y 301.106,Z 389.19,A -85,B 0,C 180,E1 -16255.932,E2 -16255.932} C_VEL
LIN {X 0,Y 299.671,Z 399.7,A -85,B 0,C 180,E1 -16260.198,E2 -16260.198} C_VEL
LIN {X 0,Y 298.654,Z 409.606,A -85,B 0,C 180,E1 -16264.192,E2 -16264.192} C_VEL
LIN {X 0,Y 297.775,Z 420.858,A -85,B 0,C 180,E1 -16268.723,E2 -16268.723} C_VEL
LIN {X 0,Y 297.746,Z 421.305,A -85,B 0,C 180,E1 -16268.857,E2 -16268.857} C_VEL
LIN {X 0,Y 298.365,Z 435.957,A -85,B 0,C 180,E1 -16269.675,E2 -16269.675} C_VEL
LIN {X 0,Y 299.006,Z 448.391,A -85,B 0,C 180,E1 -16270.623,E2 -16270.623} C_VEL
LIN {X 0,Y 299.744,Z 461.388,A -85,B 0,C 180,E1 -16271.9,E2 -16271.9} C_VEL
LIN {X 0,Y 300.245,Z 473.154,A -85,B 0,C 180,E1 -16273.337,E2 -16273.337} C_VEL
LIN {X 0,Y 299.221,Z 484.259,A -85,B 0,C 180,E1 -16275.027,E2 -16275.027} C_VEL
LIN {X 0,Y 298.512,Z 493.383,A -85,B 0,C 180,E1 -16276.729,E2 -16276.729} C_VEL
LIN {X 0,Y 297.99,Z 502.253,A -85,B 0,C 180,E1 -16278.78,E2 -16278.78} C_VEL
LIN {X 0,Y 297.827,Z 509.413,A -85,B 0,C 180,E1 -16280.835,E2 -16280.835} C_VEL
LIN {X 0,Y 297.967,Z 514.509,A -85,B 0,C 180,E1 -16282.647,E2 -16282.647} C_VEL
LIN {X 0,Y 298.203,Z 518.837,A -85,B 0,C 180,E1 -16284.59,E2 -16284.59} C_VEL
LIN {X 0,Y 298.39,Z 521.229,A -85,B 0,C 180,E1 -16285.948,E2 -16285.948} C_VEL
LIN {X 0,Y 298.529,Z 523.051,A -85,B 0,C 180,E1 -16287.301,E2 -16287.301} C_VEL
LIN {X 0,Y 298.676,Z 524.4,A -85,B 0,C 180,E1 -16288.652,E2 -16288.652} C_VEL
LIN {X 0,Y 298.88,Z 525.311,A -85,B 0,C 180,E1 -16290,E2 -16290} C_VEL
LIN {X 0,Y 298.515,Z 525.646,A -85,B 0,C 180,E1 -16291.349,E2 -16291.349} C_VEL
LIN {X 0,Y 297.888,Z 525.005,A -85,B 0,C 180,E1 -16294.059,E2 -16294.059} C_VEL
LIN {X 0,Y 297.634,Z 524.059,A -85,B 0,C 180,E1 -16295.42,E2 -16295.42} C_VEL
LIN {X 0,Y 297.356,Z 522.499,A -85,B 0,C 180,E1 -16296.94,E2 -16296.94} C_VEL
LIN {X 0,Y 297.203,Z 518.663,A -85,B 0,C 180,E1 -16299.528,E2 -16299.528} C_VEL
LIN {X 0,Y 297.529,Z 514.576,A -85,B 0,C 180,E1 -16301.583,E2 -16301.583} C_VEL
LIN {X 0,Y 298.648,Z 507.582,A -85,B 0,C 180,E1 -16304.306,E2 -16304.306} C_VEL
LIN {X 0,Y 299.995,Z 501.063,A -85,B 0,C 180,E1 -16306.327,E2 -16306.327} C_VEL
LIN {X 0,Y 302.35,Z 491.872,A -85,B 0,C 180,E1 -16308.64,E2 -16308.64} C_VEL
LIN {X 0,Y 304.815,Z 482.457,A -85,B 0,C 180,E1 -16310.586,E2 -16310.586} C_VEL
LIN {X 0,Y 306.5,Z 473.392,A -85,B 0,C 180,E1 -16312.231,E2 -16312.231} C_VEL
LIN {X 0,Y 308.55,Z 462.409,A -85,B 0,C 180,E1 -16313.944,E2 -16313.944} C_VEL
LIN {X 0,Y 309.536,Z 451.336,A -85,B 0,C 180,E1 -16315.556,E2 -16315.556} C_VEL
LIN {X 0,Y 309.437,Z 438.625,A -85,B 0,C 180,E1 -16317.371,E2 -16317.371} C_VEL
LIN {X 0,Y 308.492,Z 426.965,A -85,B 0,C 180,E1 -16319.065,E2 -16319.065} C_VEL
LIN {X 0,Y 306.586,Z 414.436,A -85,B 0,C 180,E1 -16321.017,E2 -16321.017} C_VEL
LIN {X 0,Y 305.075,Z 407.382,A -85,B 0,C 180,E1 -16322.242,E2 -16322.242} C_VEL
LIN {X 0,Y 304.057,Z 402.788,A -85,B 0,C 180,E1 -16323.079,E2 -16323.079} C_VEL
LIN {X 0,Y 303.944,Z 401.598,A -85,B 0,C 180,E1 -16323.256,E2 -16323.256} C_VEL
LIN {X 0,Y 302.389,Z 396.554,A -85,B 0,C 180,E1 -16324.352,E2 -16324.352} C_VEL
LIN {X 0,Y 302.024,Z 393.599,A -85,B 0,C 180,E1 -16324.859,E2 -16324.859} C_VEL
LIN {X 0,Y 303.984,Z 385.945,A -85,B 0,C 180,E1 -16328.626,E2 -16328.626} C_VEL
LIN {X 0,Y 303.435,Z 381.688,A -85,B 0,C 180,E1 -16331.248,E2 -16331.248} C_VEL
LIN {X 0,Y 302.645,Z 377.589,A -85,B 0,C 180,E1 -16334.16,E2 -16334.16} C_VEL
LIN {X 0,Y 301.775,Z 373.611,A -85,B 0,C 180,E1 -16337.516,E2 -16337.516} C_VEL
LIN {X 0,Y 301.068,Z 370.315,A -85,B 0,C 180,E1 -16340.929,E2 -16340.929} C_VEL
LIN {X 0,Y 300.621,Z 368.167,A -85,B 0,C 180,E1 -16343.823,E2 -16343.823} C_VEL
LIN {X 0,Y 301.549,Z 369.624,A -85,B 0,C 180,E1 -16344.659,E2 -16344.659} C_VEL
LIN {X 0,Y 304.278,Z 371.303,A -85,B 0,C 180,E1 -16346.335,E2 -16346.335} C_VEL
LIN {X 0,Y 305.694,Z 373.042,A -85,B 0,C 180,E1 -16347.25,E2 -16347.25} C_VEL
LIN {X 0,Y 306.983,Z 373.77,A -85,B 0,C 180,E1 -16347.895,E2 -16347.895} C_VEL
LIN {X 0,Y 308.361,Z 375.762,A -85,B 0,C 180,E1 -16348.736,E2 -16348.736} C_VEL
LIN {X 0,Y 309.935,Z 377.13,A -85,B 0,C 180,E1 -16349.506,E2 -16349.506} C_VEL
LIN {X 0,Y 312.838,Z 381.785,A -85,B 0,C 180,E1 -16351.182,E2 -16351.182} C_VEL
LIN {X 0,Y 316.095,Z 390.46,A -85,B 0,C 180,E1 -16353.597,E2 -16353.597} C_VEL
LIN {X 0,Y 318.092,Z 398.269,A -85,B 0,C 180,E1 -16355.582,E2 -16355.582} C_VEL
LIN {X 0,Y 318.458,Z 401.311,A -85,B 0,C 180,E1 -16356.304,E2 -16356.304} C_VEL
LIN {X 0,Y 315.507,Z 411.569,A -85,B 0,C 180,E1 -16358.092,E2 -16358.092} C_VEL
LIN {X 0,Y 312.714,Z 420.128,A -85,B 0,C 180,E1 -16359.956,E2 -16359.956} C_VEL
LIN {X 0,Y 310.148,Z 427.158,A -85,B 0,C 180,E1 -16361.845,E2 -16361.845} C_VEL
LIN {X 0,Y 307.493,Z 433.64,A -85,B 0,C 180,E1 -16364.081,E2 -16364.081} C_VEL
LIN {X 0,Y 305.587,Z 437.95,A -85,B 0,C 180,E1 -16366.026,E2 -16366.026} C_VEL
LIN {X 0,Y 303.785,Z 441.298,A -85,B 0,C 180,E1 -16367.982,E2 -16367.982} C_VEL
LIN {X 0,Y 302.804,Z 442.976,A -85,B 0,C 180,E1 -16369.299,E2 -16369.299} C_VEL
LIN {X 0,Y 301.965,Z 444.243,A -85,B 0,C 180,E1 -16370.623,E2 -16370.623} C_VEL
LIN {X 0,Y 300.46,Z 445.571,A -85,B 0,C 180,E1 -16373.283,E2 -16373.283} C_VEL
LIN {X 0,Y 299.916,Z 445.653,A -85,B 0,C 180,E1 -16374.621,E2 -16374.621} C_VEL
LIN {X 0,Y 299.44,Z 445.32,A -85,B 0,C 180,E1 -16375.962,E2 -16375.962} C_VEL
LIN {X 0,Y 298.87,Z 443.457,A -85,B 0,C 180,E1 -16378.652,E2 -16378.652} C_VEL
LIN {X 0,Y 298.761,Z 441.934,A -85,B 0,C 180,E1 -16380,E2 -16380} C_VEL
LIN {X 0,Y 298.55,Z 438.859,A -85,B 0,C 180,E1 -16382.023,E2 -16382.023} C_VEL
LIN {X 0,Y 298.384,Z 434.793,A -85,B 0,C 180,E1 -16384.052,E2 -16384.052} C_VEL
LIN {X 0,Y 298.91,Z 429.597,A -85,B 0,C 180,E1 -16386.073,E2 -16386.073} C_VEL
LIN {X 0,Y 299.366,Z 421.986,A -85,B 0,C 180,E1 -16388.437,E2 -16388.437} C_VEL
LIN {X 0,Y 300.045,Z 413.669,A -85,B 0,C 180,E1 -16390.508,E2 -16390.508} C_VEL
LIN {X 0,Y 300.734,Z 403.895,A -85,B 0,C 180,E1 -16392.484,E2 -16392.484} C_VEL
LIN {X 0,Y 301.658,Z 393.822,A -85,B 0,C 180,E1 -16394.16,E2 -16394.16} C_VEL
LIN {X 0,Y 302.542,Z 381.384,A -85,B 0,C 180,E1 -16395.84,E2 -16395.84} C_VEL
LIN {X 0,Y 302.855,Z 377.033,A -85,B 0,C 180,E1 -16396.344,E2 -16396.344} C_VEL
LIN {X 0,Y 300.312,Z 365.852,A -85,B 0,C 180,E1 -16397.596,E2 -16397.596} C_VEL
LIN {X 0,Y 298.563,Z 358.287,A -85,B 0,C 180,E1 -16398.351,E2 -16398.351} C_VEL
LIN {X 0,Y 298.432,Z 358.308,A -85,B 0,C 180,E1 -16402.135,E2 -16402.135} C_VEL
LIN {X 0,Y 298.488,Z 358.306,A -85,B 0,C 180,E1 -16405.076,E2 -16405.076} C_VEL
LIN {X 0,Y 298.466,Z 358.304,A -85,B 0,C 180,E1 -16408.095,E2 -16408.095} C_VEL
LIN {X 0,Y 298.397,Z 358.312,A -85,B 0,C 180,E1 -16412.016,E2 -16412.016} C_VEL
LIN {X 0,Y 298.434,Z 358.308,A -85,B 0,C 180,E1 -16416.067,E2 -16416.067} C_VEL
LIN {X 0,Y 298.419,Z 358.31,A -85,B 0,C 180,E1 -16419.484,E2 -16419.484} C_VEL
LIN {X 0,Y 298.432,Z 358.31,A -85,B 0,C 180,E1 -16423.11,E2 -16423.11} C_VEL
LIN {X 0,Y 298.403,Z 358.315,A -85,B 0,C 180,E1 -16426.921,E2 -16426.921} C_VEL
LIN {X 0,Y 298.416,Z 358.312,A -85,B 0,C 180,E1 -16431.003,E2 -16431.003} C_VEL
LIN {X 0,Y 298.433,Z 358.308,A -85,B 0,C 180,E1 -16433.932,E2 -16433.932} C_VEL
LIN {X 0,Y 298.394,Z 358.314,A -85,B 0,C 180,E1 -16437.984,E2 -16437.984} C_VEL
LIN {X 0,Y 298.459,Z 358.305,A -85,B 0,C 180,E1 -16441.904,E2 -16441.904} C_VEL
LIN {X 0,Y 298.486,Z 358.303,A -85,B 0,C 180,E1 -16444.924,E2 -16444.924} C_VEL
LIN {X 0,Y 298.466,Z 358.303,A -85,B 0,C 180,E1 -16449.316,E2 -16449.316} C_VEL
LIN {X 0,Y 298.539,Z 358.299,A -85,B 0,C 180,E1 -16452.179,E2 -16452.179} C_VEL
LIN {X 0,Y 298.594,Z 358.288,A -85,B 0,C 180,E1 -16454.995,E2 -16454.995} C_VEL
LIN {X 0,Y 298.592,Z 358.288,A -85,B 0,C 180,E1 -16459.147,E2 -16459.147} C_VEL
LIN {X 0,Y 298.742,Z 358.273,A -85,B 0,C 180,E1 -16461.886,E2 -16461.886} C_VEL
LIN {X 0,Y 298.658,Z 358.281,A -85,B 0,C 180,E1 -16464.599,E2 -16464.599} C_VEL
LIN {X 0,Y 298.923,Z 358.248,A -85,B 0,C 180,E1 -16468.653,E2 -16468.653} C_VEL
LIN {X 0,Y 298.925,Z 358.247,A -85,B 0,C 180,E1 -16471.347,E2 -16471.347} C_VEL
LIN {X 0,Y 298.788,Z 358.264,A -85,B 0,C 180,E1 -16476.754,E2 -16476.754} C_VEL
LIN {X 0,Y 298.636,Z 358.285,A -85,B 0,C 180,E1 -16479.482,E2 -16479.482} C_VEL
LIN {X 0,Y 298.553,Z 358.296,A -85,B 0,C 180,E1 -16483.616,E2 -16483.616} C_VEL
LIN {X 0,Y 298.55,Z 358.294,A -85,B 0,C 180,E1 -16486.409,E2 -16486.409} C_VEL
LIN {X 0,Y 298.513,Z 358.303,A -85,B 0,C 180,E1 -16489.655,E2 -16489.655} C_VEL
LIN {X 0,Y 298.458,Z 358.31,A -85,B 0,C 180,E1 -16493.598,E2 -16493.598} C_VEL
LIN {X 0,Y 298.487,Z 358.301,A -85,B 0,C 180,E1 -16496.575,E2 -16496.575} C_VEL
LIN {X 0,Y 298.417,Z 358.313,A -85,B 0,C 180,E1 -16499.642,E2 -16499.642} C_VEL
LIN {X 0,Y 298.396,Z 358.313,A -85,B 0,C 180,E1 -16502.801,E2 -16502.801} C_VEL
LIN {X 0,Y 298.467,Z 358.305,A -85,B 0,C 180,E1 -16506.813,E2 -16506.813} C_VEL
LIN {X 0,Y 298.453,Z 358.31,A -85,B 0,C 180,E1 -16511.251,E2 -16511.251} C_VEL
LIN {X 0,Y 298.418,Z 358.313,A -85,B 0,C 180,E1 -16515.047,E2 -16515.047} C_VEL
LIN {X 0,Y 298.39,Z 358.316,A -85,B 0,C 180,E1 -16518.912,E2 -16518.912} C_VEL
LIN {X 0,Y 298.446,Z 358.311,A -85,B 0,C 180,E1 -16523.193,E2 -16523.193} C_VEL
LIN {X 0,Y 298.398,Z 358.316,A -85,B 0,C 180,E1 -16527.2,E2 -16527.2} C_VEL
LIN {X 0,Y 298.435,Z 358.31,A -85,B 0,C 180,E1 -16530.615,E2 -16530.615} C_VEL
LIN {X 0,Y 298.487,Z 358.302,A -85,B 0,C 180,E1 -16533.474,E2 -16533.474} C_VEL
LIN {X 0,Y 298.439,Z 358.311,A -85,B 0,C 180,E1 -16536.697,E2 -16536.697} C_VEL
LIN {X 0,Y 298.543,Z 358.299,A -85,B 0,C 180,E1 -16540.757,E2 -16540.757} C_VEL
LIN {X 0,Y 298.597,Z 358.291,A -85,B 0,C 180,E1 -16544.995,E2 -16544.995} C_VEL
LIN {X 0,Y 298.598,Z 358.289,A -85,B 0,C 180,E1 -16549.147,E2 -16549.147} C_VEL
LIN {X 0,Y 298.763,Z 358.266,A -85,B 0,C 180,E1 -16551.886,E2 -16551.886} C_VEL
LIN {X 0,Y 298.664,Z 358.285,A -85,B 0,C 180,E1 -16554.599,E2 -16554.599} C_VEL
LIN {X 0,Y 298.927,Z 358.25,A -85,B 0,C 180,E1 -16558.653,E2 -16558.653} C_VEL
LIN {X 0,Y 298.929,Z 358.246,A -85,B 0,C 180,E1 -16561.347,E2 -16561.347} C_VEL
LIN {X 0,Y 298.653,Z 358.28,A -85,B 0,C 180,E1 -16565.35,E2 -16565.35} C_VEL
LIN {X 0,Y 298.065,Z 358.358,A -85,B 0,C 180,E1 -16566.477,E2 -16566.477} C_VEL
LIN {X 0,Y 295.216,Z 358.716,A -85,B 0,C 180,E1 -16568.31,E2 -16568.31} C_VEL
LIN {X 0,Y 292.728,Z 359.023,A -85,B 0,C 180,E1 -16569.797,E2 -16569.797} C_VEL
LIN {X 0,Y 291.628,Z 359.157,A -85,B 0,C 180,E1 -16570.951,E2 -16570.951} C_VEL
LIN {X 0,Y 291.526,Z 359.168,A -85,B 0,C 180,E1 -16571.342,E2 -16571.342} C_VEL
LIN {X 0,Y 291.559,Z 359.164,A -85,B 0,C 180,E1 -16575.376,E2 -16575.376} C_VEL
LIN {X 0,Y 291.454,Z 359.18,A -85,B 0,C 180,E1 -16579.875,E2 -16579.875} C_VEL
LIN {X 0,Y 291.404,Z 359.187,A -85,B 0,C 180,E1 -16584.205,E2 -16584.205} C_VEL
LIN {X 0,Y 291.426,Z 359.181,A -85,B 0,C 180,E1 -16587.271,E2 -16587.271} C_VEL
LIN {X 0,Y 291.341,Z 359.193,A -85,B 0,C 180,E1 -16590.437,E2 -16590.437} C_VEL
LIN {X 0,Y 291.349,Z 359.193,A -85,B 0,C 180,E1 -16593.698,E2 -16593.698} C_VEL
LIN {X 0,Y 291.397,Z 359.185,A -85,B 0,C 180,E1 -16597.259,E2 -16597.259} C_VEL
LIN {X 0,Y 291.375,Z 359.188,A -85,B 0,C 180,E1 -16600.636,E2 -16600.636} C_VEL
LIN {X 0,Y 291.405,Z 359.285,A -85,B 0,C 180,E1 -16602.104,E2 -16602.104} C_VEL
LIN {X 0,Y 292.95,Z 367.425,A -85,B 0,C 180,E1 -16606.031,E2 -16606.031} C_VEL
LIN {X 0,Y 294.636,Z 375.79,A -85,B 0,C 180,E1 -16609.906,E2 -16609.906} C_VEL
LIN {X 0,Y 295.401,Z 380.01,A -85,B 0,C 180,E1 -16611.787,E2 -16611.787} C_VEL
LIN {X 0,Y 294.503,Z 386.664,A -85,B 0,C 180,E1 -16614.612,E2 -16614.612} C_VEL
LIN {X 0,Y 292.978,Z 397.019,A -85,B 0,C 180,E1 -16618.952,E2 -16618.952} C_VEL
LIN {X 0,Y 291.671,Z 408.322,A -85,B 0,C 180,E1 -16623.65,E2 -16623.65} C_VEL
LIN {X 0,Y 290.798,Z 418.791,A -85,B 0,C 180,E1 -16628,E2 -16628} C_VEL
LIN {X 0,Y 290.699,Z 420.247,A -85,B 0,C 180,E1 -16628.598,E2 -16628.598} C_VEL
LIN {X 0,Y 291.286,Z 435.398,A -85,B 0,C 180,E1 -16629.486,E2 -16629.486} C_VEL
LIN {X 0,Y 291.943,Z 448.984,A -85,B 0,C 180,E1 -16630.578,E2 -16630.578} C_VEL
LIN {X 0,Y 292.636,Z 460.957,A -85,B 0,C 180,E1 -16631.807,E2 -16631.807} C_VEL
LIN {X 0,Y 293.157,Z 472.585,A -85,B 0,C 180,E1 -16633.281,E2 -16633.281} C_VEL
LIN {X 0,Y 292.167,Z 483.591,A -85,B 0,C 180,E1 -16635.013,E2 -16635.013} C_VEL
LIN {X 0,Y 291.468,Z 492.631,A -85,B 0,C 180,E1 -16636.758,E2 -16636.758} C_VEL
LIN {X 0,Y 290.976,Z 501.434,A -85,B 0,C 180,E1 -16638.859,E2 -16638.859} C_VEL
LIN {X 0,Y 290.821,Z 508.53,A -85,B 0,C 180,E1 -16640.962,E2 -16640.962} C_VEL
LIN {X 0,Y 291.003,Z 514.178,A -85,B 0,C 180,E1 -16643.064,E2 -16643.064} C_VEL
LIN {X 0,Y 291.338,Z 518.503,A -85,B 0,C 180,E1 -16645.157,E2 -16645.157} C_VEL
LIN {X 0,Y 291.541,Z 521.588,A -85,B 0,C 180,E1 -16647.236,E2 -16647.236} C_VEL
LIN {X 0,Y 291.695,Z 523.006,A -85,B 0,C 180,E1 -16648.619,E2 -16648.619} C_VEL
LIN {X 0,Y 291.914,Z 523.979,A -85,B 0,C 180,E1 -16650,E2 -16650} C_VEL
LIN {X 0,Y 291.496,Z 524.392,A -85,B 0,C 180,E1 -16651.381,E2 -16651.381} C_VEL
LIN {X 0,Y 291.067,Z 524.362,A -85,B 0,C 180,E1 -16652.768,E2 -16652.768} C_VEL
LIN {X 0,Y 290.832,Z 523.904,A -85,B 0,C 180,E1 -16654.157,E2 -16654.157} C_VEL
LIN {X 0,Y 290.556,Z 523.021,A -85,B 0,C 180,E1 -16655.552,E2 -16655.552} C_VEL
LIN {X 0,Y 290.306,Z 521.688,A -85,B 0,C 180,E1 -16656.988,E2 -16656.988} C_VEL
LIN {X 0,Y 290.131,Z 517.916,A -85,B 0,C 180,E1 -16659.762,E2 -16659.762} C_VEL
LIN {X 0,Y 290.535,Z 513.995,A -85,B 0,C 180,E1 -16661.865,E2 -16661.865} C_VEL
LIN {X 0,Y 291.741,Z 507.215,A -85,B 0,C 180,E1 -16664.652,E2 -16664.652} C_VEL
LIN {X 0,Y 292.644,Z 502.865,A -85,B 0,C 180,E1 -16666.131,E2 -16666.131} C_VEL
LIN {X 0,Y 294.832,Z 494.801,A -85,B 0,C 180,E1 -16668.412,E2 -16668.412} C_VEL
LIN {X 0,Y 297.798,Z 484.669,A -85,B 0,C 180,E1 -16670.732,E2 -16670.732} C_VEL
